	{attribute 'TcIecLibraryType'}
	{attribute 'external_name' := 'F_VN_CreateStaModel_GUID_E1160B26_F7CF_4D94_F7D4_A5AFD71C214D'}
	(* Create a Simplified TopoART neural network of the specified type. The initial reference count is set to one if a new model is created and kept, otherwise. Models of this type support on-line training (sample by sample), retraining, as well as scalar and vectorial predictions. It requires all input except class labels (i.e., samples and training outputs/predictions) to lie in the interval [0.0, 1.0]. The predictions of regressors need to be rescaled from the interval [0.0, 1.0] to their respective value range before usage. Depending on the parameter settings and the number of available training samples, repeated training with the same data may improve the results. Like other neural networks based on the Adaptive Resonance Theory (ART), Simplified TopoART neural networks are not prone to catastrophic inference and patricularly well-suited to incremental learning tasks. *)
	FUNCTION F_VN_CreateStaModel : HRESULT
	VAR_INPUT
		ipMlModel	:	REFERENCE TO ITcVnMlModel;	(* Returns the created model (Non-zero interface pointers are reused.) *)
		eStaType	:	ETcVnSta;	(* Simpified TopoART model type *)
		fRho	:	LREAL;	(* Vigilance parameter (controls the number of neurons that are inserted and the maximum size of the formed categories; valid range: [0.0, 1.0]; suggested range: [0.8, 1.0)) *)
		hrPrev	:	HRESULT;	(* HRESULT indicating the result of previous operations (If SUCCEEDED(hrPrev) equals false, no operation is executed.) *)
	END_VAR

END_FUNCTION

// Functions/Machine Learning/F_VN_CreateStaModelExp

	{attribute 'TcIecLibraryType'}
	{attribute 'external_name' := 'F_VN_CreateStaModelExp_GUID_8FBAA2F4_0437_4354_E26E_F8E69F80A9C2'}
	(* Create a Simplified TopoART neural network of the specified type. The initial reference count is set to one if a new model is created and kept, otherwise. Models of this type support on-line training (sample by sample), retraining, as well as scalar and vectorial predictions. It requires all input except class labels (i.e., samples and training outputs/predictions) to lie in the interval [0.0, 1.0]. The predictions of regressors need to be rescaled from the interval [0.0, 1.0] to their respective value range before usage. Depending on the parameter settings and the number of available training samples, repeated training with the same data may improve the results. Like other neural networks based on the Adaptive Resonance Theory (ART), Simplified TopoART neural networks are not prone to catastrophic inference and patricularly well-suited to incremental learning tasks. (expert function) *)
	FUNCTION F_VN_CreateStaModelExp : HRESULT
	VAR_INPUT
		ipMlModel	:	REFERENCE TO ITcVnMlModel;	(* Returns the created model (Non-zero interface pointers are reused.) *)
		eStaType	:	ETcVnSta;	(* Simpified TopoART model type *)
		fRho	:	LREAL;	(* Vigilance parameter (controls the number of neurons that are inserted and the maximum size of the formed categories; valid range: [0.0, 1.0]; suggested range: [0.8, 1.0)) *)
		nNu	:	UDINT;	(* Number of neurons used for classification and prediction (must be larger than or equal to 1; suggested range: [1, 10); default: 3) *)
		bDoublePrecision	:	BOOL;	(* If true, the model is generated with double precision (LREAL) instead of single precision (REAL). (default: FALSE) *)
		hrPrev	:	HRESULT;	(* HRESULT indicating the result of previous operations (If SUCCEEDED(hrPrev) equals false, no operation is executed.) *)
	END_VAR

END_FUNCTION

// Functions/Machine Learning/F_VN_CreateStaModelExp2

	{attribute 'TcIecLibraryType'}
	{attribute 'external_name' := 'F_VN_CreateStaModelExp2_GUID_332943B0_2083_4579_FA51_A2E1DF860F25'}
	(* Create a Simplified TopoART neural network of the specified type. The initial reference count is set to one if a new model is created and kept, otherwise. Models of this type support on-line training (sample by sample), retraining, as well as scalar and vectorial predictions. It requires all input except class labels (i.e., samples and training outputs/predictions) to lie in the interval [0.0, 1.0]. The predictions of regressors need to be rescaled from the interval [0.0, 1.0] to their respective value range before usage. Depending on the parameter settings and the number of available training samples, repeated training with the same data may improve the results. Like other neural networks based on the Adaptive Resonance Theory (ART), Simplified TopoART neural networks are not prone to catastrophic inference and patricularly well-suited to incremental learning tasks. (additional expert function providing parameters for fine-tuning and noise reduction) *)
	FUNCTION F_VN_CreateStaModelExp2 : HRESULT
	VAR_INPUT
		ipMlModel	:	REFERENCE TO ITcVnMlModel;	(* Returns the created model (Non-zero interface pointers are reused.) *)
		eStaType	:	ETcVnSta;	(* Simpified TopoART model type *)
		fRho	:	LREAL;	(* Vigilance parameter (controls the number of neurons that are inserted and the maximum size of the formed categories; valid range: [0.0, 1.0]; suggested range: [0.8, 1.0)) *)
		nNu	:	UDINT;	(* Number of neurons used for classification and prediction (must be larger than or equal to 1; suggested range: [1, 10); default: 3) *)
		bDoublePrecision	:	BOOL;	(* If true, the model is generated with double precision (LREAL) instead of single precision (REAL). (default: FALSE) *)
		fBetaSbm	:	LREAL;	(* Learning rate of the second best-matching neuron (learning the second best-matching neuron keeps related categories closer together and might improve the results but may require a higher number of neurons and training runs; a value of 0.0 disables learning of the second best-matching neuron; valid range: [0.0, 1.0]; suggested range: [0.0, 0.5]); default: 0.0 *)
		nPhi	:	UDINT;	(* Number of samples a neuron must have learnt to become permanent (required for noise reduction; works in conjunction with nTau; must be larger than or equal to 1; higher values intensify noise reduction; a value of 1 disables removal of neuron candidates; default: 1) *)
		nTau	:	UDINT;	(* Number of learning steps after which node removal is performed (required for noise reduction; works in conjunction with nPhi; must be large enough to allow neuron candidates representing non-noise samples to become the best-matching neuron at least nPhi times before node removal; default: 100) *)
		hrPrev	:	HRESULT;	(* HRESULT indicating the result of previous operations (If SUCCEEDED(hrPrev) equals false, no operation is executed.) *)
	END_VAR

END_FUNCTION

// Functions/Machine Learning/F_VN_CreateSvmModel

	{attribute 'TcIecLibraryType'}
	{attribute 'external_name' := 'F_VN_CreateSvmModel_GUID_897BE96D_4F53_4CE0_D9B9_89EE3A81129D'}
	(* Create an SVM model of the specified type. The initial reference count is set to one if a new model is created and kept, otherwise. Models of this type neither support on-line training (sample by sample) nor retraining. Predictions can only be scalar. *)
	FUNCTION F_VN_CreateSvmModel : HRESULT
	VAR_INPUT
		ipMlModel	:	REFERENCE TO ITcVnMlModel;	(* Returns the created model (Non-zero interface pointers are reused.) *)
		eSvmType	:	ETcVnSvm;	(* SVM model type *)
		fC	:	LREAL;	(* Parameter C (required for TCVN_SVM_C_CLASSIFIER, TCVN_SVM_EPS_REGRESSOR, and TCVN_SVM_NU_REGRESSOR; ignored otherwise) *)
		fNu	:	LREAL;	(* Parameter nu (required for TCVN_SVM_NU_CLASSIFIER, TCVN_SVM_NOVELTY_DETECTOR, and TCVN_SVM_NU_REGRESSOR; ignored otherwise) *)
		fP	:	LREAL;	(* Parameter p (required for TCVN_SVM_EPS_REGRESSOR; ignored otherwise) *)
		eKernelType	:	ETcVnSvmKernelType;	(* Kernel type *)
		fGamma	:	LREAL;	(* Parameter gamma (used by polynomial, RBF, sigmoid, and chi-squared kernels; ignored otherwise) *)
		fCoef0	:	LREAL;	(* parameter coef0 (used by polynomial and sigmoid kernels; ignored otherwise) *)
		fDegree	:	LREAL;	(* Degree (used by polynomial kernels; ignored otherwise) *)
		hrPrev	:	HRESULT;	(* HRESULT indicating the result of previous operations (If SUCCEEDED(hrPrev) equals false, no operation is executed.) *)
	END_VAR

END_FUNCTION

// Functions/Machine Learning/F_VN_CreateSvmModelExp

	{attribute 'TcIecLibraryType'}
	{attribute 'external_name' := 'F_VN_CreateSvmModelExp_GUID_846E7362_1CAD_446F_E876_9CE57F3D46D8'}
	(* Create an SVM model of the specified type. The initial reference count is set to one if a new model is created and kept, otherwise. Models of this type neither support on-line training (sample by sample) nor retraining. Predictions can only be scalar. (expert function) *)
	FUNCTION F_VN_CreateSvmModelExp : HRESULT
	VAR_INPUT
		ipMlModel	:	REFERENCE TO ITcVnMlModel;	(* Returns the created model (Non-zero interface pointers are reused.) *)
		eSvmType	:	ETcVnSvm;	(* SVM model type *)
		fC	:	LREAL;	(* Parameter C (required for TCVN_SVM_C_CLASSIFIER, TCVN_SVM_EPS_REGRESSOR, and TCVN_SVM_NU_REGRESSOR; ignored otherwise) *)
		fNu	:	LREAL;	(* Parameter nu (required for TCVN_SVM_NU_CLASSIFIER, TCVN_SVM_NOVELTY_DETECTOR, and TCVN_SVM_NU_REGRESSOR; ignored otherwise) *)
		fP	:	LREAL;	(* Parameter p (required for TCVN_SVM_EPS_REGRESSOR; ignored otherwise) *)
		eKernelType	:	ETcVnSvmKernelType;	(* Kernel type *)
		fGamma	:	LREAL;	(* Parameter gamma (used by polynomial, RBF, sigmoid, and chi-squared kernels; ignored otherwise) *)
		fCoef0	:	LREAL;	(* Parameter coef0 (used by polynomial and sigmoid kernels; ignored otherwise) *)
		fDegree	:	LREAL;	(* Degree (used by polynomial kernels; ignored otherwise) *)
		nMaxIterations	:	UDINT;	(* Maximum number of iterations (disabled if it equals 0 and fEpsilon is different from 0.0; triggers the usage of the default value of 100000 if nMaxIterations and fEpsilon equal 0) *)
		fEpsilon	:	LREAL;	(* Maximum allowed difference of the error between two successive iterations (disabled if it equals 0.0 and nMaxIterations is different from 0; triggers the usage of the default value of 0.00001 if nMaxIterations and fEpsilon equal 0) *)
		hrPrev	:	HRESULT;	(* HRESULT indicating the result of previous operations (If SUCCEEDED(hrPrev) equals false, no operation is executed.) *)
	END_VAR

END_FUNCTION

// Functions/Machine Learning/F_VN_CreateSvmModelExp2

	{attribute 'TcIecLibraryType'}
	{attribute 'external_name' := 'F_VN_CreateSvmModelExp2_GUID_80A60ED2_EC58_4E94_FB00_9F02BF868F8D'}
	(* Create an SVM model of the specified type. The initial reference count is set to one if a new model is created and kept, otherwise. Models of this type neither support on-line training (sample by sample) nor retraining. Predictions can only be scalar. (additional expert function for C support vector classifiers) *)
	FUNCTION F_VN_CreateSvmModelExp2 : HRESULT
	VAR_INPUT
		ipMlModel	:	REFERENCE TO ITcVnMlModel;	(* Returns the created model (Non-zero interface pointers are reused.) *)
		eSvmType	:	ETcVnSvm;	(* SVM model type *)
		fC	:	LREAL;	(* Parameter C (required for TCVN_SVM_C_CLASSIFIER, TCVN_SVM_EPS_REGRESSOR, and TCVN_SVM_NU_REGRESSOR; ignored otherwise) *)
		fNu	:	LREAL;	(* Parameter nu (required for TCVN_SVM_NU_CLASSIFIER, TCVN_SVM_NOVELTY_DETECTOR, and TCVN_SVM_NU_REGRESSOR; ignored otherwise) *)
		fP	:	LREAL;	(* Parameter p (required for TCVN_SVM_EPS_REGRESSOR; ignored otherwise) *)
		eKernelType	:	ETcVnSvmKernelType;	(* Kernel type *)
		fGamma	:	LREAL;	(* Parameter gamma (used by polynomial, RBF, sigmoid, and chi-squared kernels; ignored otherwise) *)
		fCoef0	:	LREAL;	(* Parameter coef0 (used by polynomial and sigmoid kernels; ignored otherwise) *)
		fDegree	:	LREAL;	(* Degree (used by polynomial kernels; ignored otherwise) *)
		nMaxIterations	:	UDINT;	(* Maximum number of iterations (disabled if it equals 0 and fEpsilon is different from 0.0; triggers the usage of the default value of 100000 if nMaxIterations and fEpsilon equal 0) *)
		fEpsilon	:	LREAL;	(* Maximum allowed difference of the error between two successive iterations (disabled if it equals 0.0 and nMaxIterations is different from 0; triggers the usage of the default value of 0.00001 if nMaxIterations and fEpsilon equal 0) *)
		ipClassWeights	:	ITcVnContainer;	(* Class weights (ContainerType_Vector_REAL or ContainerType_Vector_LREAL; only valid if eSvmType equals TCVN_SVM_C_CLASSIFIER; optional, set to 0 if not required or not allowed; default: 0) *)
		hrPrev	:	HRESULT;	(* HRESULT indicating the result of previous operations (If SUCCEEDED(hrPrev) equals false, no operation is executed.) *)
	END_VAR

END_FUNCTION

// Functions/Machine Learning/F_VN_CreateSvmSgdClassifier

	{attribute 'TcIecLibraryType'}
	{attribute 'external_name' := 'F_VN_CreateSvmSgdClassifier_GUID_269DD8EF_015C_48A4_C0CA_F5AB46B04256'}
	(* Create a linear SVM classifier using stochastic gradient descent for training. The initial reference count is set to one if a new model is created and kept, otherwise. This SVM classifier is only applicable to binary classification problems. It learns a separating hyperplane between a class with label -1 and a class with label 1. These class labels are predefined. For training, any positive class labels are mapped to 1 and any negative class labels are mapped to -1. Models of this type neither support on-line training (sample by sample) nor retraining. *)
	FUNCTION F_VN_CreateSvmSgdClassifier : HRESULT
	VAR_INPUT
		ipMlModel	:	REFERENCE TO ITcVnMlModel;	(* Returns the created model (Non-zero interface pointers are reused.) *)
		hrPrev	:	HRESULT;	(* HRESULT indicating the result of previous operations (If SUCCEEDED(hrPrev) equals false, no operation is executed.) *)
	END_VAR

END_FUNCTION

// Functions/Machine Learning/F_VN_CreateSvmSgdClassifierExp

	{attribute 'TcIecLibraryType'}
	{attribute 'external_name' := 'F_VN_CreateSvmSgdClassifierExp_GUID_DA02D1B9_7AEC_4B7E_EFA9_4DE4F7562F76'}
	(* Create a linear SVM classifier using stochastic gradient descent for training. The initial reference count is set to one if a new model is created and kept, otherwise. This SVM classifier is only applicable to binary classification problems. It learns a separating hyperplane between a class with label -1 and a class with label 1. These class labels are predefined. For training, any positive class labels are mapped to 1 and any negative class labels are mapped to -1. Models of this type neither support on-line training (sample by sample) nor retraining. (expert function) *)
	FUNCTION F_VN_CreateSvmSgdClassifierExp : HRESULT
	VAR_INPUT
		ipMlModel	:	REFERENCE TO ITcVnMlModel;	(* Returns the created model (Non-zero interface pointers are reused.) *)
		eType	:	ETcVnSvmSgdClassifierType;	(* Learning algorithm type (default: TCVN_SSCT_ASGD) *)
		eMarginType	:	ETcVnSvmSgdClassifierMarginType;	(* Margin type (default: TCVN_SSCMT_SOFT_MARGIN) *)
		fMarginRegularization	:	REAL;	(* Margin regularization parameter (default: 0.00001) *)
		fInitialStepSize	:	REAL;	(* Initial step size (default: 0.05) *)
		fStepDecreasingPower	:	REAL;	(* Power parameter (default: 0.75) *)
		nMaxIterations	:	UDINT;	(* Maximum number of iterations (disabled if it equals 0 and fEpsilon is different from 0.0; triggers the usage of the default value of 100000 if nMaxIterations and fEpsilon equal 0) *)
		fEpsilon	:	LREAL;	(* Maximum allowed difference of the error between two successive iterations (disabled if it equals 0.0 and nMaxIterations is different from 0; triggers the usage of the default value of 0.00001 if nMaxIterations and fEpsilon equal 0) *)
		hrPrev	:	HRESULT;	(* HRESULT indicating the result of previous operations (If SUCCEEDED(hrPrev) equals false, no operation is executed.) *)
	END_VAR

END_FUNCTION

// Functions/Machine Learning/F_VN_FeatureTransform

	{attribute 'TcIecLibraryType'}
	{attribute 'external_name' := 'F_VN_FeatureTransform_GUID_2974563E_7A4B_46F8_CDD5_2C6660AA8677'}
	(* Apply a feature transform to one or more sample(s). *)
	FUNCTION F_VN_FeatureTransform : HRESULT
	VAR_INPUT
		ipFeatureTransform	:	ITcVnMlModel;	(* Feature transform instance to be used *)
		ipSamples	:	ITcUnknown;	(* Container holding one or more of input sample(s) (ContainerType_Vector_REAL, ContainerType_Vector_LREAL, ContainerType_Vector_Vector_REAL, or ContainerType_Vector_Vector_LREAL) *)
		pipTransformed	:	POINTER TO ITcUnknown;	(* Returns the transformed sample(s) using the same type like ipSamples *)
		hrPrev	:	HRESULT;	(* HRESULT indicating the result of previous operations (If SUCCEEDED(hrPrev) equals false, no operation is executed.) *)
	END_VAR

END_FUNCTION

// Functions/Machine Learning/F_VN_GetBatchClusters

	{attribute 'TcIecLibraryType'}
	{attribute 'external_name' := 'F_VN_GetBatchClusters_GUID_BDFDD55D_49E0_4ED4_F9D7_56F0B43B3AD1'}
	(* Get the IDs of the best-matching clusters of a batch of samples. *)
	FUNCTION F_VN_GetBatchClusters : HRESULT
	VAR_INPUT
		ipClusterer	:	ITcVnMlModel;	(* Clusterer to be used *)
		ipSamples	:	ITcUnknown;	(* Container holding a batch of input samples (ContainerType_Vector_Vector_REAL or ContainerType_Vector_Vector_LREAL) *)
		ipClusters	:	REFERENCE TO ITcVnContainer;	(* Returns the cluster IDs (ContainerType_Vector_DINT) *)
		hrPrev	:	HRESULT;	(* HRESULT indicating the result of previous operations (If SUCCEEDED(hrPrev) equals false, no operation is executed.) *)
	END_VAR

END_FUNCTION

// Functions/Machine Learning/F_VN_GetBatchClustersExp

	{attribute 'TcIecLibraryType'}
	{attribute 'external_name' := 'F_VN_GetBatchClustersExp_GUID_05544234_9673_4981_C2EB_ED06839AEAC5'}
	(* Get the IDs of the best-matching clusters of a batch of samples. *)
	FUNCTION F_VN_GetBatchClustersExp : HRESULT
	VAR_INPUT
		ipClusterer	:	ITcVnMlModel;	(* Clusterer to be used *)
		ipSamples	:	ITcUnknown;	(* Container holding a batch of input samples (ContainerType_Vector_Vector_REAL or ContainerType_Vector_Vector_LREAL) *)
		ipClusters	:	REFERENCE TO ITcVnContainer;	(* Returns the cluster IDs (ContainerType_Vector_DINT) *)
		ipNovelties	:	REFERENCE TO ITcVnContainer;	(* Returns the degree of novelty (0.0 if a sample is completely known; > 0.0 otherwise) of each sample (ContainerType_Vector_REAL; optional, set to 0 if not required) *)
		hrPrev	:	HRESULT;	(* HRESULT indicating the result of previous operations (If SUCCEEDED(hrPrev) equals false, no operation is executed.) *)
	END_VAR

END_FUNCTION

// Functions/Machine Learning/F_VN_GetBatchNovelties

	{attribute 'TcIecLibraryType'}
	{attribute 'external_name' := 'F_VN_GetBatchNovelties_GUID_93485253_723B_43D7_F5BA_82F42BF1627D'}
	(* Get the degree of novelty of multiple samples. *)
	FUNCTION F_VN_GetBatchNovelties : HRESULT
	VAR_INPUT
		ipNoveltyDetector	:	ITcVnMlModel;	(* Novelty detector to be used *)
		ipSamples	:	ITcUnknown;	(* Container holding a batch of input samples (ContainerType_Vector_Vector_REAL or ContainerType_Vector_Vector_LREAL) *)
		ipNovelties	:	REFERENCE TO ITcVnContainer;	(* Returns the degree of novelty (0.0 if a sample is completely known; > 0.0 otherwise) of each sample (ContainerType_Vector_REAL) *)
		hrPrev	:	HRESULT;	(* HRESULT indicating the result of previous operations (If SUCCEEDED(hrPrev) equals false, no operation is executed.) *)
	END_VAR

END_FUNCTION

// Functions/Machine Learning/F_VN_GetClusterCenter

	{attribute 'TcIecLibraryType'}
	{attribute 'external_name' := 'F_VN_GetClusterCenter_GUID_E0FF4273_E499_42E6_FD8B_B6C189318933'}
	(* Get the center of a cluster. *)
	FUNCTION F_VN_GetClusterCenter : HRESULT
	VAR_INPUT
		ipClusterer	:	ITcVnMlModel;	(* Clusterer to be used *)
		nCluster	:	DINT;	(* Cluster ID of the cluster the center of which is requested *)
		ipCenter	:	REFERENCE TO ITcVnContainer;	(* Returns the cluster center (ContainerType_Vector_REAL or ContainerType_Vector_LREAL depending on the floating point type internally used by the clusterer) *)
		hrPrev	:	HRESULT;	(* HRESULT indicating the result of previous operations (If SUCCEEDED(hrPrev) equals false, no operation is executed.) *)
	END_VAR

END_FUNCTION

// Functions/Machine Learning/F_VN_GetClusterNum

	{attribute 'TcIecLibraryType'}
	{attribute 'external_name' := 'F_VN_GetClusterNum_GUID_BBFC8079_9A14_4919_DF9B_189A17F3D8B0'}
	(* Get the number of clusters used by this clusterer. *)
	FUNCTION F_VN_GetClusterNum : HRESULT
	VAR_INPUT
		ipClusterer	:	ITcVnMlModel;	(* Clusterer to be used *)
	END_VAR
	VAR_IN_OUT
		nClusterNum	:	ULINT;	(* Returns the number of clusters *)
	END_VAR
	VAR_INPUT
		hrPrev	:	HRESULT;	(* HRESULT indicating the result of previous operations (If SUCCEEDED(hrPrev) equals false, no operation is executed.) *)
	END_VAR

END_FUNCTION

// Functions/Machine Learning/F_VN_GetFeatureScales

	{attribute 'TcIecLibraryType'}
	{attribute 'external_name' := 'F_VN_GetFeatureScales_GUID_11456483_F148_42D1_FF0B_C79EBE00E4BF'}
	(* Calculate the scaling parameters for each feature in the input samples based on the scaling type. *)
	FUNCTION F_VN_GetFeatureScales : HRESULT
	VAR_INPUT
		ipSamples	:	ITcVnContainer;	(* Container holding input sample(s) (ContainerType_Vector_REAL, ContainerType_Vector_LREAL, ContainerType_Vector_Vector_REAL or ContainerType_Vector_Vector_LREAL) *)
		ipScales	:	REFERENCE TO ITcVnContainer;	(* Returns a container with the scaling parameters for each feature (Vector_REAL or Vector_LREAL depending on the type of ipSamples). *)
		eFeatureScalingType	:	ETcVnFeatureScalingType;	(* Feature scaling type *)
		hrPrev	:	HRESULT;	(* HRESULT indicating the result of previous operations (If SUCCEEDED(hrPrev) equals false, no operation is executed.) *)
	END_VAR

END_FUNCTION

// Functions/Machine Learning/F_VN_GetSampleCluster

	{attribute 'TcIecLibraryType'}
	{attribute 'external_name' := 'F_VN_GetSampleCluster_GUID_DD81FA91_6080_4B4C_E0CB_06C1EA1FBF26'}
	(* Get the ID of the best-matching cluster of a single sample. *)
	FUNCTION F_VN_GetSampleCluster : HRESULT
	VAR_INPUT
		ipClusterer	:	ITcVnMlModel;	(* Clusterer to be used *)
		ipSample	:	ITcUnknown;	(* Container holding a single input sample (ContainerType_Vector_REAL or ContainerType_Vector_LREAL) *)
	END_VAR
	VAR_IN_OUT
		nCluster	:	DINT;	(* Returns the ID of the cluster the sample has been assigned to *)
	END_VAR
	VAR_INPUT
		hrPrev	:	HRESULT;	(* HRESULT indicating the result of previous operations (If SUCCEEDED(hrPrev) equals false, no operation is executed.) *)
	END_VAR

END_FUNCTION

// Functions/Machine Learning/F_VN_GetSampleClusterExp

	{attribute 'TcIecLibraryType'}
	{attribute 'external_name' := 'F_VN_GetSampleClusterExp_GUID_DB048C2F_2D45_4057_FF4A_13B0418E387B'}
	(* Get the ID of the best-matching cluster of a single sample. (expert function) *)
	FUNCTION F_VN_GetSampleClusterExp : HRESULT
	VAR_INPUT
		ipClusterer	:	ITcVnMlModel;	(* Clusterer to be used *)
		ipSample	:	ITcUnknown;	(* Container holding a single input sample (ContainerType_Vector_REAL or ContainerType_Vector_LREAL) *)
	END_VAR
	VAR_IN_OUT
		nCluster	:	DINT;	(* Returns the ID of the cluster the sample has been assigned to *)
	END_VAR
	VAR_INPUT
		fNovelty	:	REFERENCE TO REAL;	(* Returns the degree of novelty (0.0 if a sample is completely known; > 0.0 otherwise) of the presented sample (optional, set to 0 if not required) *)
		hrPrev	:	HRESULT;	(* HRESULT indicating the result of previous operations (If SUCCEEDED(hrPrev) equals false, no operation is executed.) *)
	END_VAR

END_FUNCTION

// Functions/Machine Learning/F_VN_GetSampleNovelty

	{attribute 'TcIecLibraryType'}
	{attribute 'external_name' := 'F_VN_GetSampleNovelty_GUID_3DC424A1_B05C_4823_FDDB_8F0CF1505A59'}
	(* Get the degree of novelty of a single sample. *)
	FUNCTION F_VN_GetSampleNovelty : HRESULT
	VAR_INPUT
		ipNoveltyDetector	:	ITcVnMlModel;	(* Novelty detector to be used *)
		ipSample	:	ITcUnknown;	(* Container holding a single input sample (ContainerType_Vector_REAL or ContainerType_Vector_LREAL) *)
	END_VAR
	VAR_IN_OUT
		fNovelty	:	REAL;	(* Returns the degree of novelty (0.0 if a sample is completely known; > 0.0 otherwise) of the presented sample *)
	END_VAR
	VAR_INPUT
		hrPrev	:	HRESULT;	(* HRESULT indicating the result of previous operations (If SUCCEEDED(hrPrev) equals false, no operation is executed.) *)
	END_VAR

END_FUNCTION

// Functions/Machine Learning/F_VN_InverseFeatureScaling

	{attribute 'TcIecLibraryType'}
	{attribute 'external_name' := 'F_VN_InverseFeatureScaling_GUID_FAE38955_0DF9_4C1B_F986_91CF8149BAD2'}
	(* Apply the inverse of feature scaling to one or more sample(s). *)
	FUNCTION F_VN_InverseFeatureScaling : HRESULT
	VAR_INPUT
		ipSamples	:	ITcVnContainer;	(* Container holding one or more input sample(s) (ContainerType_Vector_REAL, ContainerType_Vector_LREAL, ContainerType_Vector_Vector_REAL, or ContainerType_Vector_Vector_LREAL) *)
		ipScales	:	ITcVnContainer;	(* Container with the scaling parameters of each feature (type ContainerType_Vector_REAL or ContainerType_Vector_LREAL). *)
		ipInverseSamples	:	REFERENCE TO ITcVnContainer;	(* Returns the inversed sample(s) using the scaling type and parameters of ipScales. It has the same type of ipSamples. If the same container ipSamples is used, the source data will be replaced. *)
		hrPrev	:	HRESULT;	(* HRESULT indicating the result of previous operations (If SUCCEEDED(hrPrev) equals false, no operation is executed.) *)
	END_VAR

END_FUNCTION

// Functions/Machine Learning/F_VN_InverseFeatureScaling_REAL

	{attribute 'TcIecLibraryType'}
	{attribute 'external_name' := 'F_VN_InverseFeatureScaling_REAL_GUID_166D968F_147A_4210_E12A_96ABB8210FC5'}
	(* Apply the inverse of feature scaling to a single value. *)
	FUNCTION F_VN_InverseFeatureScaling_REAL : HRESULT
	VAR_INPUT
		fSample	:	REAL;	(* Sample value *)
		ipScales	:	ITcVnContainer;	(* Container with the scaling parameters of each feature (type ContainerType_Vector_REAL or ContainerType_Vector_LREAL). *)
	END_VAR
	VAR_IN_OUT
		fInverseSample	:	REAL;	(* Returns the inversed sample. *)
	END_VAR
	VAR_INPUT
		hrPrev	:	HRESULT;	(* HRESULT indicating the result of previous operations (If SUCCEEDED(hrPrev) equals false, no operation is executed.) *)
	END_VAR

END_FUNCTION

// Functions/Machine Learning/F_VN_InverseFeatureScalingExp

	{attribute 'TcIecLibraryType'}
	{attribute 'external_name' := 'F_VN_InverseFeatureScalingExp_GUID_647DF1EC_D563_4098_CB76_97CF9047029E'}
	(* Apply the inverse of feature scaling to one or more sample(s). [fA, fB] should be used if the scaling has been performed using TCVN_FST1_MINMAX with a predetermined output range.. (expert function) *)
	FUNCTION F_VN_InverseFeatureScalingExp : HRESULT
	VAR_INPUT
		ipSamples	:	ITcVnContainer;	(* Container holding one or more input sample(s) (ContainerType_Vector_REAL, ContainerType_Vector_LREAL, ContainerType_Vector_Vector_REAL, or ContainerType_Vector_Vector_LREAL) *)
		ipScales	:	ITcVnContainer;	(* Container with the scaling parameters of each feature (type ContainerType_Vector_REAL or ContainerType_Vector_LREAL). *)
		ipInverseSamples	:	REFERENCE TO ITcVnContainer;	(* Returns the inversed sample(s) using the scaling type and parameters of ipScales. It has the same type of ipSamples. If the same container ipSamples is used, the source data will be replaced. *)
		fA	:	LREAL;	(* represents the lower bound of the range for TCVN_FST1_MINMAX *)
		fB	:	LREAL;	(* represents the upper bound of the range for TCVN_FST1_MINMAX *)
		hrPrev	:	HRESULT;	(* HRESULT indicating the result of previous operations (If SUCCEEDED(hrPrev) equals false, no operation is executed.) *)
	END_VAR

END_FUNCTION

// Functions/Machine Learning/F_VN_InverseFeatureScalingExp_REAL

	{attribute 'TcIecLibraryType'}
	{attribute 'external_name' := 'F_VN_InverseFeatureScalingExp_REAL_GUID_CDDB6A41_2C3B_42C5_C560_BF34481C5C25'}
	(* Apply the inverse of feature scaling to a single value. [fA, fB] should be used if the scaling has been performed using TCVN_FST1_MINMAX with a predetermined output range. *)
	FUNCTION F_VN_InverseFeatureScalingExp_REAL : HRESULT
	VAR_INPUT
		fSample	:	REAL;	(* Sample value *)
		ipScales	:	ITcVnContainer;	(* Container with the scaling parameters of each feature (type ContainerType_Vector_REAL or ContainerType_Vector_LREAL). *)
	END_VAR
	VAR_IN_OUT
		fInverseSample	:	REAL;	(* Returns the inversed sample. *)
	END_VAR
	VAR_INPUT
		fA	:	LREAL;	(* represents the lower bound of the range for TCVN_FST1_MINMAX *)
		fB	:	LREAL;	(* represents the upper bound of the range for TCVN_FST1_MINMAX *)
		hrPrev	:	HRESULT;	(* HRESULT indicating the result of previous operations (If SUCCEEDED(hrPrev) equals false, no operation is executed.) *)
	END_VAR

END_FUNCTION

// Functions/Machine Learning/F_VN_InverseFeatureTransform

	{attribute 'TcIecLibraryType'}
	{attribute 'external_name' := 'F_VN_InverseFeatureTransform_GUID_329639C8_477F_4462_EC9B_877837D05181'}
	(* Apply an inverse feature transform to one or more sample(s). *)
	FUNCTION F_VN_InverseFeatureTransform : HRESULT
	VAR_INPUT
		ipFeatureTransform	:	ITcVnMlModel;	(* Feature transform instance to be used *)
		ipSamples	:	ITcUnknown;	(* Container holding one or more of input sample(s) (ContainerType_Vector_REAL, ContainerType_Vector_LREAL, ContainerType_Vector_Vector_REAL, or ContainerType_Vector_Vector_LREAL) *)
		pipTransformed	:	POINTER TO ITcUnknown;	(* Returns the transformed sample(s) using the same type like ipSamples *)
		hrPrev	:	HRESULT;	(* HRESULT indicating the result of previous operations (If SUCCEEDED(hrPrev) equals false, no operation is executed.) *)
	END_VAR

END_FUNCTION

// Functions/Machine Learning/F_VN_PredictBatch

	{attribute 'TcIecLibraryType'}
	{attribute 'external_name' := 'F_VN_PredictBatch_GUID_7906A2A4_9C1A_4EB4_C744_43C3CB5A8C79'}
	(* Compute predictions for a batch of samples. *)
	FUNCTION F_VN_PredictBatch : HRESULT
	VAR_INPUT
		ipMlModel	:	ITcVnMlModel;	(* Classifier or regressor to be used *)
		ipSamples	:	ITcUnknown;	(* Container holding a batch of input samples (ContainerType_Vector_Vector_REAL or ContainerType_Vector_Vector_LREAL) *)
		ipPredictions	:	REFERENCE TO ITcVnContainer;	(* Returns the predicted outputs (depending on ipSamples; class labels (for classification, ContainerType_Vector_DINT) or real-valued predictions (for regression with scalar output, ContainerType_Vector_REAL or ContainerType_Vector_LREAL; for regression with vectorial output, ContainerType_Vector_Vector_REAL or ContainerType_Vector_Vector_LREAL)) *)
		hrPrev	:	HRESULT;	(* HRESULT indicating the result of previous operations (If SUCCEEDED(hrPrev) equals false, no operation is executed.) *)
	END_VAR

END_FUNCTION

// Functions/Machine Learning/F_VN_PredictBatchExp

	{attribute 'TcIecLibraryType'}
	{attribute 'external_name' := 'F_VN_PredictBatchExp_GUID_C7E3B96F_60A8_4AAD_F208_9E382A2099F8'}
	(* Compute predictions for a batch of samples. (expert function) *)
	FUNCTION F_VN_PredictBatchExp : HRESULT
	VAR_INPUT
		ipMlModel	:	ITcVnMlModel;	(* Classifier or regressor to be used *)
		ipSamples	:	ITcUnknown;	(* Container holding a batch of input samples (ContainerType_Vector_Vector_REAL or ContainerType_Vector_Vector_LREAL) *)
		ipPredictions	:	REFERENCE TO ITcVnContainer;	(* Returns the predicted outputs (depending on ipSamples; class labels (for classification, ContainerType_Vector_DINT) or real-valued predictions (for regression with scalar output, ContainerType_Vector_REAL or ContainerType_Vector_LREAL; for regression with vectorial output, ContainerType_Vector_Vector_REAL or ContainerType_Vector_Vector_LREAL)) *)
		ipNovelties	:	REFERENCE TO ITcVnContainer;	(* Returns the degree of novelty (0.0 if a sample is completely known; > 0.0 otherwise) of each sample (ContainerType_Vector_REAL; optional, set to 0 if not required) *)
		hrPrev	:	HRESULT;	(* HRESULT indicating the result of previous operations (If SUCCEEDED(hrPrev) equals false, no operation is executed.) *)
	END_VAR

END_FUNCTION

// Functions/Machine Learning/F_VN_PredictSampleClass

	{attribute 'TcIecLibraryType'}
	{attribute 'external_name' := 'F_VN_PredictSampleClass_GUID_4A7121E2_C40C_4D6B_D87B_86DF80F92135'}
	(* Classify a single sample. *)
	FUNCTION F_VN_PredictSampleClass : HRESULT
	VAR_INPUT
		ipClassifier	:	ITcVnMlModel;	(* Classifier to be used *)
		ipSample	:	ITcUnknown;	(* Container holding a single input sample (ContainerType_Vector_REAL or ContainerType_Vector_LREAL) *)
	END_VAR
	VAR_IN_OUT
		nClass	:	DINT;	(* Returns the classification result *)
	END_VAR
	VAR_INPUT
		hrPrev	:	HRESULT;	(* HRESULT indicating the result of previous operations (If SUCCEEDED(hrPrev) equals false, no operation is executed.) *)
	END_VAR

END_FUNCTION

// Functions/Machine Learning/F_VN_PredictSampleClassExp

	{attribute 'TcIecLibraryType'}
	{attribute 'external_name' := 'F_VN_PredictSampleClassExp_GUID_7E949930_4452_469B_E4D3_CE540860A53A'}
	(* Classify a single sample. (expert function) *)
	FUNCTION F_VN_PredictSampleClassExp : HRESULT
	VAR_INPUT
		ipClassifier	:	ITcVnMlModel;	(* Classifier to be used *)
		ipSample	:	ITcUnknown;	(* Container holding a single input sample (ContainerType_Vector_REAL or ContainerType_Vector_LREAL) *)
	END_VAR
	VAR_IN_OUT
		nClass	:	DINT;	(* Returns the classification result *)
	END_VAR
	VAR_INPUT
		fNovelty	:	REFERENCE TO REAL;	(* Returns the degree of novelty (0.0 if a sample is completely known; > 0.0 otherwise) of the presented sample (optional, set to 0 if not required) *)
		hrPrev	:	HRESULT;	(* HRESULT indicating the result of previous operations (If SUCCEEDED(hrPrev) equals false, no operation is executed.) *)
	END_VAR

END_FUNCTION

// Functions/Machine Learning/F_VN_PredictSampleScalar

	{attribute 'TcIecLibraryType'}
	{attribute 'external_name' := 'F_VN_PredictSampleScalar_GUID_A40A5FE6_578F_494C_E511_207CF80FE52D'}
	(* Compute a scalar prediction for a single sample. *)
	FUNCTION F_VN_PredictSampleScalar : HRESULT
	VAR_INPUT
		ipRegressor	:	ITcVnMlModel;	(* Regressor to be used *)
		ipSample	:	ITcUnknown;	(* Container holding a single input sample (ContainerType_Vector_REAL or ContainerType_Vector_LREAL) *)
	END_VAR
	VAR_IN_OUT
		fPrediction	:	REAL;	(* Returns the predicted output *)
	END_VAR
	VAR_INPUT
		hrPrev	:	HRESULT;	(* HRESULT indicating the result of previous operations (If SUCCEEDED(hrPrev) equals false, no operation is executed.) *)
	END_VAR

END_FUNCTION

// Functions/Machine Learning/F_VN_PredictSampleScalarExp

	{attribute 'TcIecLibraryType'}
	{attribute 'external_name' := 'F_VN_PredictSampleScalarExp_GUID_367E34F1_4772_4005_C610_209F58792692'}
	(* Compute a scalar prediction for a single sample. (expert function) *)
	FUNCTION F_VN_PredictSampleScalarExp : HRESULT
	VAR_INPUT
		ipRegressor	:	ITcVnMlModel;	(* Regressor to be used *)
		ipSample	:	ITcUnknown;	(* Container holding a single input sample (ContainerType_Vector_REAL or ContainerType_Vector_LREAL) *)
	END_VAR
	VAR_IN_OUT
		fPrediction	:	REAL;	(* Returns the predicted output *)
	END_VAR
	VAR_INPUT
		fNovelty	:	REFERENCE TO REAL;	(* Returns the degree of novelty (0.0 if a sample is completely known; > 0.0 otherwise) of the presented sample (optional, set to 0 if not required) *)
		hrPrev	:	HRESULT;	(* HRESULT indicating the result of previous operations (If SUCCEEDED(hrPrev) equals false, no operation is executed.) *)
	END_VAR

END_FUNCTION

// Functions/Machine Learning/F_VN_PredictSampleVector

	{attribute 'TcIecLibraryType'}
	{attribute 'external_name' := 'F_VN_PredictSampleVector_GUID_172DA4F7_FC29_4D5D_F84B_CCD2E6CC2758'}
	(* Compute a vectorial prediction for a single sample. *)
	FUNCTION F_VN_PredictSampleVector : HRESULT
	VAR_INPUT
		ipRegressor	:	ITcVnMlModel;	(* Regressor to be used *)
		ipSample	:	ITcUnknown;	(* Container holding a single input sample (ContainerType_Vector_REAL or ContainerType_Vector_LREAL) *)
		ipPrediction	:	REFERENCE TO ITcVnContainer;	(* Returns the predicted output (ContainerType_Vector_REAL or ContainerType_Vector_LREAL, depending on ipSample) *)
		hrPrev	:	HRESULT;	(* HRESULT indicating the result of previous operations (If SUCCEEDED(hrPrev) equals false, no operation is executed.) *)
	END_VAR

END_FUNCTION

// Functions/Machine Learning/F_VN_PredictSampleVectorExp

	{attribute 'TcIecLibraryType'}
	{attribute 'external_name' := 'F_VN_PredictSampleVectorExp_GUID_07735102_4AA2_46A6_C4D9_B15C63AD99B2'}
	(* Compute a vectorial prediction for a single sample. (expert function) *)
	FUNCTION F_VN_PredictSampleVectorExp : HRESULT
	VAR_INPUT
		ipRegressor	:	ITcVnMlModel;	(* Regressor to be used *)
		ipSample	:	ITcUnknown;	(* Container holding a single input sample (ContainerType_Vector_REAL or ContainerType_Vector_LREAL) *)
		ipPrediction	:	REFERENCE TO ITcVnContainer;	(* Returns the predicted output (ContainerType_Vector_REAL or ContainerType_Vector_LREAL, depending on ipSample) *)
		fNovelty	:	REFERENCE TO REAL;	(* Returns the degree of novelty (0.0 if a sample is completely known; > 0.0 otherwise) of the presented sample (optional, set to 0 if not required) *)
		hrPrev	:	HRESULT;	(* HRESULT indicating the result of previous operations (If SUCCEEDED(hrPrev) equals false, no operation is executed.) *)
	END_VAR

END_FUNCTION

// Functions/Machine Learning/F_VN_FeatureScaling

	{attribute 'TcIecLibraryType'}
	{attribute 'external_name' := 'F_VN_FeatureScaling_GUID_9FB5D54E_2B28_4BDC_DFDE_B62044F088AC'}
	(* Apply a feature scaling to one or more sample(s). *)
	FUNCTION F_VN_FeatureScaling : HRESULT
	VAR_INPUT
		ipSamples	:	ITcVnContainer;	(* Container holding one or more input sample(s) (ContainerType_Vector_REAL, ContainerType_Vector_LREAL, ContainerType_Vector_Vector_REAL, or ContainerType_Vector_Vector_LREAL) *)
		ipScales	:	ITcVnContainer;	(* Container with the scaling parameters of each feature (type ContainerType_Vector_REAL or ContainerType_Vector_LREAL). *)
		ipScaledSamples	:	REFERENCE TO ITcVnContainer;	(* Returns the scaled sample(s) using the same type like ipSamples. If the same container ipSamples is uesd, the source data will be replaced. *)
		hrPrev	:	HRESULT;	(* HRESULT indicating the result of previous operations (If SUCCEEDED(hrPrev) equals false, no operation is executed.) *)
	END_VAR

END_FUNCTION

// Functions/Machine Learning/F_VN_FeatureScalingExp

	{attribute 'TcIecLibraryType'}
	{attribute 'external_name' := 'F_VN_FeatureScalingExp_GUID_66B24BFE_9031_4553_F21F_FA0BBFFFF2B0'}
	(* Apply a feature scaling to one or more sample(s) and get output range between [fA, fB] in the case of TCVN_FST1_MINMAX.  (expert function) *)
	FUNCTION F_VN_FeatureScalingExp : HRESULT
	VAR_INPUT
		ipSamples	:	ITcVnContainer;	(* Container holding one or more input sample(s) (ContainerType_Vector_REAL, ContainerType_Vector_LREAL, ContainerType_Vector_Vector_REAL, or ContainerType_Vector_Vector_LREAL) *)
		ipScales	:	ITcVnContainer;	(* Container with the scaling parameters of each feature (type ContainerType_Vector_REAL or ContainerType_Vector_LREAL). *)
		ipScaledSamples	:	REFERENCE TO ITcVnContainer;	(* Returns the scaled sample(s) using the same type like ipSamples. If the same container ipSamples is uesd, the source data will be replaced. *)
		fA	:	LREAL;	(* represents the lower bound of the range for TCVN_FST1_MINMAX *)
		fB	:	LREAL;	(* represents the upper bound of the range for TCVN_FST1_MINMAX *)
		hrPrev	:	HRESULT;	(* HRESULT indicating the result of previous operations (If SUCCEEDED(hrPrev) equals false, no operation is executed.) *)
	END_VAR

END_FUNCTION

// Functions/Machine Learning/F_VN_TrainBatch

	{attribute 'TcIecLibraryType'}
	{attribute 'external_name' := 'F_VN_TrainBatch_GUID_73F82A21_79CD_4474_CA00_DD7E810BA348'}
	(* Train a classifier, a clusterer, a novelty detector, or a regressor with a batch of samples. On-line trainable models are trained once with each sample. Depending on the application and the number of available training samples, repeated training of such models with the same data may improve the results. *)
	FUNCTION F_VN_TrainBatch : HRESULT
	VAR_INPUT
		ipMlModel	:	ITcVnMlModel;	(* Classifier, clusterer, novelty detector, or regressor to be used *)
		ipSamples	:	ITcUnknown;	(* Container holding a batch of input samples (ContainerType_Vector_Vector_REAL or ContainerType_Vector_Vector_LREAL) *)
		ipOutputs	:	ITcVnContainer;	(* Class labels (for classification, ContainerType_Vector_DINT) or target outputs (for regression with scalar output, ContainerType_Vector_REAL or ContainerType_Vector_LREAL; for regression with vectorial output, ContainerType_Vector_Vector_REAL or ContainerType_Vector_Vector_LREAL) to be learnt (must be 0 for clusterers and for novelty detectors) *)
		hrPrev	:	HRESULT;	(* HRESULT indicating the result of previous operations (If SUCCEEDED(hrPrev) equals false, no operation is executed.) *)
	END_VAR

END_FUNCTION

// Functions/Machine Learning/F_VN_TrainBatchClusters

	{attribute 'TcIecLibraryType'}
	{attribute 'external_name' := 'F_VN_TrainBatchClusters_GUID_272ADC4A_55CD_40B4_F968_65B14199D4F5'}
	(* Train a clusterer with a batch of samples and return the IDs of the clusters the samples have been assigned to, if requested. On-line trainable clusterers are trained once with each sample. Depending on the application and the number of available training samples, repeated training of such models with the same data may improve the results. *)
	FUNCTION F_VN_TrainBatchClusters : HRESULT
	VAR_INPUT
		ipClusterer	:	ITcVnMlModel;	(* Clusterer to be used *)
		ipSamples	:	ITcUnknown;	(* Container holding a batch of input samples (ContainerType_Vector_Vector_REAL or ContainerType_Vector_Vector_LREAL) *)
		ipClusters	:	REFERENCE TO ITcVnContainer;	(* Returns the IDs of the clusters the samples have been assigned to (ContainerType_Vector_DINT; optional, set to 0 if not required) *)
		hrPrev	:	HRESULT;	(* HRESULT indicating the result of previous operations (If SUCCEEDED(hrPrev) equals false, no operation is executed.) *)
	END_VAR

END_FUNCTION

// Functions/Machine Learning/F_VN_TrainSample

	{attribute 'TcIecLibraryType'}
	{attribute 'external_name' := 'F_VN_TrainSample_GUID_6F6670E1_3692_44BE_FB06_674C6EFB3F43'}
	(* Train a clusterer or a novelty detector with a single sample. *)
	FUNCTION F_VN_TrainSample : HRESULT
	VAR_INPUT
		ipMlModel	:	ITcVnMlModel;	(* Clusterer or novelty detector to be used *)
		ipSample	:	ITcUnknown;	(* Container holding a single input sample (ContainerType_Vector_REAL or ContainerType_Vector_LREAL) *)
		hrPrev	:	HRESULT;	(* HRESULT indicating the result of previous operations (If SUCCEEDED(hrPrev) equals false, no operation is executed.) *)
	END_VAR

END_FUNCTION

// Functions/Machine Learning/F_VN_TrainSampleClass

	{attribute 'TcIecLibraryType'}
	{attribute 'external_name' := 'F_VN_TrainSampleClass_GUID_05A64E90_55FA_45CF_FDB8_2105F78E81D1'}
	(* Train a classifier with a single sample. *)
	FUNCTION F_VN_TrainSampleClass : HRESULT
	VAR_INPUT
		ipClassifier	:	ITcVnMlModel;	(* Classifier to be used *)
		ipSample	:	ITcUnknown;	(* Container holding a single input sample (ContainerType_Vector_REAL or ContainerType_Vector_LREAL) *)
		nClass	:	DINT;	(* Class label to be learnt *)
		hrPrev	:	HRESULT;	(* HRESULT indicating the result of previous operations (If SUCCEEDED(hrPrev) equals false, no operation is executed.) *)
	END_VAR

END_FUNCTION

// Functions/Machine Learning/F_VN_TrainSampleCluster

	{attribute 'TcIecLibraryType'}
	{attribute 'external_name' := 'F_VN_TrainSampleCluster_GUID_343E64C2_DE56_4145_F502_F352497DB18B'}
	(* Train a clusterer with a single sample and return the ID of the cluster the sample has been assigned to, if requested. The clusterer must be online trainable. *)
	FUNCTION F_VN_TrainSampleCluster : HRESULT
	VAR_INPUT
		ipClusterer	:	ITcVnMlModel;	(* Clusterer to be used *)
		ipSample	:	ITcUnknown;	(* Container holding a single input sample (ContainerType_Vector_REAL or ContainerType_Vector_LREAL) *)
		nCluster	:	REFERENCE TO DINT;	(* Returns the ID of the cluster the sample has been assigned to (If the pointer is 0, no cluster ID is requested.) *)
		hrPrev	:	HRESULT;	(* HRESULT indicating the result of previous operations (If SUCCEEDED(hrPrev) equals false, no operation is executed.) *)
	END_VAR

END_FUNCTION

// Functions/Machine Learning/F_VN_TrainSampleScalar

	{attribute 'TcIecLibraryType'}
	{attribute 'external_name' := 'F_VN_TrainSampleScalar_GUID_5CBD0285_80B0_4A96_F720_162C311C1FF3'}
	(* Train a regressor with a single sample and scalar output. *)
	FUNCTION F_VN_TrainSampleScalar : HRESULT
	VAR_INPUT
		ipRegressor	:	ITcVnMlModel;	(* Regressor to be used *)
		ipSample	:	ITcUnknown;	(* Container holding a single input sample (ContainerType_Vector_REAL or ContainerType_Vector_LREAL) *)
		fOutput	:	REAL;	(* Scalar output to be learnt *)
		hrPrev	:	HRESULT;	(* HRESULT indicating the result of previous operations (If SUCCEEDED(hrPrev) equals false, no operation is executed.) *)
	END_VAR

END_FUNCTION

// Functions/Machine Learning/F_VN_TrainSampleVector

	{attribute 'TcIecLibraryType'}
	{attribute 'external_name' := 'F_VN_TrainSampleVector_GUID_A5E64EDC_AD34_41AF_FAB6_19C619D724B8'}
	(* Train a regressor with a single sample and vectorial output. *)
	FUNCTION F_VN_TrainSampleVector : HRESULT
	VAR_INPUT
		ipRegressor	:	ITcVnMlModel;	(* Regressor to be used *)
		ipSample	:	ITcUnknown;	(* Container holding a single input sample (ContainerType_Vector_REAL or ContainerType_Vector_LREAL) *)
		ipOutput	:	ITcVnContainer;	(* Vectorial output to be learnt (ContainerType_Vector_REAL or ContainerType_Vector_LREAL) *)
		hrPrev	:	HRESULT;	(* HRESULT indicating the result of previous operations (If SUCCEEDED(hrPrev) equals false, no operation is executed.) *)
	END_VAR

END_FUNCTION

// Functions/Drawing/F_VN_DrawArrow

	{attribute 'TcIecLibraryType'}
	{attribute 'external_name' := 'F_VN_DrawArrow_GUID_219FAA59_40C2_4064_C408_565BDDFC528F'}
	(* Draw an arrowed line. *)
	FUNCTION F_VN_DrawArrow : HRESULT
	VAR_INPUT
		nX1	:	UDINT;	(* x coordinate of the start point *)
		nY1	:	UDINT;	(* y coordinate of the start point *)
		nX2	:	UDINT;	(* x coordinate of the end point *)
		nY2	:	UDINT;	(* y coordinate of the end point *)
		ipDestImage	:	ITcVnImage;	(* Destination image *)
	END_VAR
	VAR_IN_OUT
		aColor	:	TcVnVector4_LREAL;	(* Color *)
	END_VAR
	VAR_INPUT
		nThickness	:	DINT;	(* Line thickness *)
		bDoubleHead	:	BOOL;	(* To draw an arrow on each side of the line. *)
		hrPrev	:	HRESULT;	(* HRESULT indicating the result of previous operations (If SUCCEEDED(hrPrev) equals false, no operation is executed.) *)
	END_VAR

END_FUNCTION

// Functions/Drawing/F_VN_DrawArrow_TcVnVector4_DINT

	{attribute 'TcIecLibraryType'}
	{attribute 'external_name' := 'F_VN_DrawArrow_TcVnVector4_DINT_GUID_CD974053_3A84_4A78_FF52_9525307415ED'}
	(* Draw an arrowed line. *)
	FUNCTION F_VN_DrawArrow_TcVnVector4_DINT : HRESULT
	VAR_IN_OUT
		aLine	:	TcVnVector4_DINT;	(* The start and end point of a line segment [x1, y1, x2, y2] *)
	END_VAR
	VAR_INPUT
		ipDestImage	:	ITcVnImage;	(* Destination image *)
	END_VAR
	VAR_IN_OUT
		aColor	:	TcVnVector4_LREAL;	(* Color *)
	END_VAR
	VAR_INPUT
		nThickness	:	DINT;	(* Line thickness *)
		bDoubleHead	:	BOOL;	(* To draw an arrow on each side of the line. *)
		hrPrev	:	HRESULT;	(* HRESULT indicating the result of previous operations (If SUCCEEDED(hrPrev) equals false, no operation is executed.) *)
	END_VAR

END_FUNCTION

// Functions/Drawing/F_VN_DrawArrowExp

	{attribute 'TcIecLibraryType'}
	{attribute 'external_name' := 'F_VN_DrawArrowExp_GUID_9874EFD7_9D2C_4A6E_E29C_9A7DCBDB5A42'}
	(* Draws an arrowed line. (expert function) *)
	FUNCTION F_VN_DrawArrowExp : HRESULT
	VAR_INPUT
		nX1	:	UDINT;	(* x coordinate of the start point *)
		nY1	:	UDINT;	(* y coordinate of the start point *)
		nX2	:	UDINT;	(* x coordinate of the end point *)
		nY2	:	UDINT;	(* y coordinate of the end point *)
		ipDestImage	:	ITcVnImage;	(* Destination image *)
	END_VAR
	VAR_IN_OUT
		aColor	:	TcVnVector4_LREAL;	(* Color *)
	END_VAR
	VAR_INPUT
		nThickness	:	DINT;	(* Line thickness *)
		bDoubleHead	:	BOOL;	(* To draw an arrow on each side of the line. *)
		eLineType	:	ETcVnLineType;	(* Line type *)
		nShift	:	UDINT;	(* Fractional bits of the coordinates (bit shift) *)
		fTipLenght	:	LREAL;	(* Lenght of the arrow's tip as a fraction of the line's lenght *)
		hrPrev	:	HRESULT;	(* HRESULT indicating the result of previous operations (If SUCCEEDED(hrPrev) equals false, no operation is executed.) *)
	END_VAR

END_FUNCTION

// Functions/Drawing/F_VN_DrawArrowExp_TcVnVector4_DINT

	{attribute 'TcIecLibraryType'}
	{attribute 'external_name' := 'F_VN_DrawArrowExp_TcVnVector4_DINT_GUID_EB1F5363_59BE_442A_FA36_95178B47EBDC'}
	(* Draws an arrowed line. (expert function) *)
	FUNCTION F_VN_DrawArrowExp_TcVnVector4_DINT : HRESULT
	VAR_IN_OUT
		aLine	:	TcVnVector4_DINT;	(* The start and end point of a line segment [x1, y1, x2, y2] *)
	END_VAR
	VAR_INPUT
		ipDestImage	:	ITcVnImage;	(* Destination image *)
	END_VAR
	VAR_IN_OUT
		aColor	:	TcVnVector4_LREAL;	(* Color *)
	END_VAR
	VAR_INPUT
		nThickness	:	DINT;	(* Line thickness *)
		bDoubleHead	:	BOOL;	(* To draw an arrow on each side of the line. *)
		eLineType	:	ETcVnLineType;	(* Line type *)
		nShift	:	UDINT;	(* Fractional bits of the coordinates (bit shift) *)
		fTipLenght	:	LREAL;	(* Lenght of the arrow's tip as a fraction of the line's lenght *)
		hrPrev	:	HRESULT;	(* HRESULT indicating the result of previous operations (If SUCCEEDED(hrPrev) equals false, no operation is executed.) *)
	END_VAR

END_FUNCTION

// Functions/Drawing/F_VN_DrawCircle

	{attribute 'TcIecLibraryType'}
	{attribute 'external_name' := 'F_VN_DrawCircle_GUID_E54EF870_255A_4D91_CCEB_101D0778E80E'}
	(* Draws a circle. *)
	FUNCTION F_VN_DrawCircle : HRESULT
	VAR_INPUT
		nCenterX	:	UDINT;	(* x coordinate of the center *)
		nCenterY	:	UDINT;	(* y coordinate of the center *)
		nRadius	:	UDINT;	(* Radius *)
		ipDestImage	:	ITcVnImage;	(* Destination image *)
	END_VAR
	VAR_IN_OUT
		aColor	:	TcVnVector4_LREAL;	(* Color *)
	END_VAR
	VAR_INPUT
		nThickness	:	DINT;	(* Line thickness (if negative, the circle is filled) *)
		hrPrev	:	HRESULT;	(* HRESULT indicating the result of previous operations (If SUCCEEDED(hrPrev) equals false, no operation is executed.) *)
	END_VAR

END_FUNCTION

// Functions/Drawing/F_VN_DrawCircleExp

	{attribute 'TcIecLibraryType'}
	{attribute 'external_name' := 'F_VN_DrawCircleExp_GUID_EBF1C3F3_0B87_4735_E6BF_D00B09B46DB9'}
	(* Draws a circle. *)
	FUNCTION F_VN_DrawCircleExp : HRESULT
	VAR_INPUT
		nCenterX	:	UDINT;	(* x coordinate of the center *)
		nCenterY	:	UDINT;	(* y coordinate of the center *)
		nRadius	:	UDINT;	(* Radius *)
		ipDestImage	:	ITcVnImage;	(* Destination image *)
	END_VAR
	VAR_IN_OUT
		aColor	:	TcVnVector4_LREAL;	(* Color *)
	END_VAR
	VAR_INPUT
		nThickness	:	DINT;	(* Line thickness (if negative, the circle is filled) *)
		eLineType	:	ETcVnLineType;	(* Line type *)
		hrPrev	:	HRESULT;	(* HRESULT indicating the result of previous operations (If SUCCEEDED(hrPrev) equals false, no operation is executed.) *)
	END_VAR

END_FUNCTION

// Functions/Drawing/F_VN_DrawCircles

	{attribute 'TcIecLibraryType'}
	{attribute 'external_name' := 'F_VN_DrawCircles_GUID_13EAF35C_B06F_4815_C884_30D225E98417'}
	(* Draws circles. *)
	FUNCTION F_VN_DrawCircles : HRESULT
	VAR_INPUT
		ipCircles	:	ITcVnContainer;	(* Container with circles (ContainerType_Vector_TcVnVector3_REAL; Each container element contains the x coordinate of the circle center [0], the y coordinate of the circle center [1], and the radius [2].) *)
		nCircleIndex	:	DINT;	(* Index of a specific circle to be drawn (if negative, all circles within the container are drawn) *)
		ipDestImage	:	ITcVnImage;	(* Destination image *)
	END_VAR
	VAR_IN_OUT
		aColor	:	TcVnVector4_LREAL;	(* Color *)
	END_VAR
	VAR_INPUT
		nThickness	:	DINT;	(* Line thickness (if negative, the circle is filled) *)
		hrPrev	:	HRESULT;	(* HRESULT indicating the result of previous operations (If SUCCEEDED(hrPrev) equals false, no operation is executed.) *)
	END_VAR

END_FUNCTION

// Functions/Drawing/F_VN_DrawCirclesExp

	{attribute 'TcIecLibraryType'}
	{attribute 'external_name' := 'F_VN_DrawCirclesExp_GUID_4084C455_AE24_4B16_CD21_E442AAEA2A01'}
	(* Draws circles. (expert function) *)
	FUNCTION F_VN_DrawCirclesExp : HRESULT
	VAR_INPUT
		ipCircles	:	ITcVnContainer;	(* Container with circles (ContainerType_Vector_TcVnVector3_REAL; Each container element contains the x coordinate of the circle center [0], the y coordinate of the circle center [1], and the radius [2].) *)
		nCircleIndex	:	DINT;	(* Index of a specific circle to be drawn (if negative, all circles within the container are drawn) *)
		ipDestImage	:	ITcVnImage;	(* Destination image *)
	END_VAR
	VAR_IN_OUT
		aColor	:	TcVnVector4_LREAL;	(* Color *)
	END_VAR
	VAR_INPUT
		nThickness	:	DINT;	(* Line thickness (if negative, the circle is filled) *)
		eLineType	:	ETcVnLineType;	(* Line type *)
		hrPrev	:	HRESULT;	(* HRESULT indicating the result of previous operations (If SUCCEEDED(hrPrev) equals false, no operation is executed.) *)
	END_VAR

END_FUNCTION

// Functions/Drawing/F_VN_DrawCircularArc

	{attribute 'TcIecLibraryType'}
	{attribute 'external_name' := 'F_VN_DrawCircularArc_GUID_E25A37E1_93AB_4946_DDE0_DA467037DDBC'}
	(* Draws a circular arc. *)
	FUNCTION F_VN_DrawCircularArc : HRESULT
	VAR_IN_OUT
		stCircularArc	:	TcVnCircularArc;	(* Circular arc definition *)
	END_VAR
	VAR_INPUT
		ipDestImage	:	ITcVnImage;	(* Destination image *)
	END_VAR
	VAR_IN_OUT
		aColor	:	TcVnVector4_LREAL;	(* Color *)
	END_VAR
	VAR_INPUT
		nThickness	:	DINT;	(* Line thickness (if negative, the arc is filled) *)
		hrPrev	:	HRESULT;	(* HRESULT indicating the result of previous operations (If SUCCEEDED(hrPrev) equals false, no operation is executed.) *)
	END_VAR

END_FUNCTION

// Functions/Drawing/F_VN_DrawCircularArcExp

	{attribute 'TcIecLibraryType'}
	{attribute 'external_name' := 'F_VN_DrawCircularArcExp_GUID_D9B37CB2_BAE4_440C_C152_969A4B69D972'}
	(* Draws a circular arc. (expert function) *)
	FUNCTION F_VN_DrawCircularArcExp : HRESULT
	VAR_IN_OUT
		stCircularArc	:	TcVnCircularArc;	(* Circular arc definition *)
	END_VAR
	VAR_INPUT
		ipDestImage	:	ITcVnImage;	(* Destination image *)
	END_VAR
	VAR_IN_OUT
		aColor	:	TcVnVector4_LREAL;	(* Color *)
	END_VAR
	VAR_INPUT
		nThickness	:	DINT;	(* Line thickness (if negative, the arc is filled) *)
		eLineType	:	ETcVnLineType;	(* Line type *)
		hrPrev	:	HRESULT;	(* HRESULT indicating the result of previous operations (If SUCCEEDED(hrPrev) equals false, no operation is executed.) *)
	END_VAR

END_FUNCTION

// Functions/Drawing/F_VN_DrawComponents

	{attribute 'TcIecLibraryType'}
	{attribute 'external_name' := 'F_VN_DrawComponents_GUID_E9922499_BF1D_45AC_D80D_6B3535350DD3'}
	(* Draw the results of connected component function. *)
	FUNCTION F_VN_DrawComponents : HRESULT
	VAR_INPUT
		ipLabelImage	:	ITcVnImage;	(* Image contains labels for each pixel (1 channel DINT or UINT). *)
		nLabelID	:	DINT;	(* Value of a specific label to be drawn (if negative, all components within the image are drawn) *)
		ipDestImage	:	REFERENCE TO ITcVnImage;	(* Destination image (An appropriate image will be created if required. The output image is 1 or 3 channels USINT). *)
		bShowLabelID	:	BOOL;	(* Show label ID in the center of the component on the destination image *)
		hrPrev	:	HRESULT;	(* HRESULT indicating the result of previous operations (If SUCCEEDED(hrPrev) equals false, no operation is executed.) *)
	END_VAR

END_FUNCTION

// Functions/Drawing/F_VN_DrawComponentsExp

	{attribute 'TcIecLibraryType'}
	{attribute 'external_name' := 'F_VN_DrawComponentsExp_GUID_67F7A137_6C61_4D22_D78F_645CEAAA63A6'}
	(* Draw the results of connected component function. (expert function) *)
	FUNCTION F_VN_DrawComponentsExp : HRESULT
	VAR_INPUT
		ipLabelImage	:	ITcVnImage;	(* Image contains labels for each pixel (1 channel DINT or UINT). *)
		nLabelID	:	DINT;	(* Value of a specific label to be drawn (if negative, all components within the image are drawn) *)
		ipDestImage	:	REFERENCE TO ITcVnImage;	(* Destination image (An appropriate image will be created if required. The output image is 1 or 3 channels USINT). *)
		bShowLabelID	:	BOOL;	(* Show lable ID in the center of the component on the destination image *)
	END_VAR
	VAR_IN_OUT
		aColor	:	TcVnVector4_LREAL;	(* Color to draw the components (for {-1, -1, -1, -1}, a random color is chosen for each component) *)
	END_VAR
	VAR_INPUT
		nThickness	:	DINT;	(* Text line thickness *)
		fFontScale	:	LREAL;	(* Scaling factor for the text *)
		hrPrev	:	HRESULT;	(* HRESULT indicating the result of previous operations (If SUCCEEDED(hrPrev) equals false, no operation is executed.) *)
	END_VAR

END_FUNCTION

// Functions/Drawing/F_VN_DrawContours

	{attribute 'TcIecLibraryType'}
	{attribute 'external_name' := 'F_VN_DrawContours_GUID_BD96A0E1_088D_495C_DC88_0A1555E00AA4'}
	(* Draws a single point set or multiple point sets that are interpreted as contours. *)
	FUNCTION F_VN_DrawContours : HRESULT
	VAR_INPUT
		ipContours	:	ITcVnContainer;	(* Single contour (ContainerType_Vector_TcVnPoint2_DINT) or multiple contours (ContainerType_Vector_Vector_TcVnPoint2_DINT) *)
		nContourIndex	:	DINT;	(* Index of a specific contour to be drawn (if negative, all contours within the container are drawn) *)
		ipDestImage	:	ITcVnImage;	(* Destination image *)
	END_VAR
	VAR_IN_OUT
		aColor	:	TcVnVector4_LREAL;	(* Color *)
	END_VAR
	VAR_INPUT
		nThickness	:	DINT;	(* Line thickness (if negative, the contours are filled) *)
		hrPrev	:	HRESULT;	(* HRESULT indicating the result of previous operations (If SUCCEEDED(hrPrev) equals false, no operation is executed.) *)
	END_VAR

END_FUNCTION

// Functions/Drawing/F_VN_DrawContoursExp

	{attribute 'TcIecLibraryType'}
	{attribute 'external_name' := 'F_VN_DrawContoursExp_GUID_CEFBF024_BBCC_4DBE_C01D_8D086DC8267C'}
	(* Draws a single point set or multiple point sets that are interpreted as contours. (expert function) *)
	FUNCTION F_VN_DrawContoursExp : HRESULT
	VAR_INPUT
		ipContours	:	ITcVnContainer;	(* Single contour (ContainerType_Vector_TcVnPoint2_DINT) or multiple contours (ContainerType_Vector_Vector_TcVnPoint2_DINT) *)
		nContourIndex	:	DINT;	(* Index of a specific contour to be drawn (if negative, all contours within the container are drawn) *)
		ipDestImage	:	ITcVnImage;	(* Destination image *)
	END_VAR
	VAR_IN_OUT
		aColor	:	TcVnVector4_LREAL;	(* Color *)
	END_VAR
	VAR_INPUT
		nThickness	:	DINT;	(* Line thickness (if negative, the contours are filled) *)
		eLineType	:	ETcVnLineType;	(* Line type *)
		ipHierarchy	:	ITcVnContainer;	(* Contour hierarchy (ContainerType_Vector_TcVnVector4_DINT) *)
		nMaxLevel	:	DINT;	(* Maximum level of contours to be drawn *)
	END_VAR
	VAR_IN_OUT
		aOffset	:	TcVnPoint;	(* Offset by which every contour point is shifted *)
	END_VAR
	VAR_INPUT
		hrPrev	:	HRESULT;	(* HRESULT indicating the result of previous operations (If SUCCEEDED(hrPrev) equals false, no operation is executed.) *)
	END_VAR

END_FUNCTION

// Functions/Drawing/F_VN_DrawEllipse

	{attribute 'TcIecLibraryType'}
	{attribute 'external_name' := 'F_VN_DrawEllipse_GUID_348B0EA6_8D61_4699_CBAC_E9971A365AF6'}
	(* Draws an ellipse. *)
	FUNCTION F_VN_DrawEllipse : HRESULT
	VAR_IN_OUT
		stEllipse	:	TcVnRotatedRectangle;	(* Ellipse to be drawn (rotation angle in degrees) *)
	END_VAR
	VAR_INPUT
		ipDestImage	:	ITcVnImage;	(* Destination image *)
	END_VAR
	VAR_IN_OUT
		aColor	:	TcVnVector4_LREAL;	(* Color *)
	END_VAR
	VAR_INPUT
		nThickness	:	DINT;	(* Line thickness (if negative, the ellipse is filled) *)
		hrPrev	:	HRESULT;	(* HRESULT indicating the result of previous operations (If SUCCEEDED(hrPrev) equals false, no operation is executed.) *)
	END_VAR

END_FUNCTION

// Functions/Drawing/F_VN_DrawEllipseExp

	{attribute 'TcIecLibraryType'}
	{attribute 'external_name' := 'F_VN_DrawEllipseExp_GUID_C5879EEA_4F57_40F1_ED9B_B7DB43373126'}
	(* Draws an ellipse. (expert function) *)
	FUNCTION F_VN_DrawEllipseExp : HRESULT
	VAR_IN_OUT
		stEllipse	:	TcVnRotatedRectangle;	(* Ellipse to be drawn (rotation angle in degrees) *)
	END_VAR
	VAR_INPUT
		ipDestImage	:	ITcVnImage;	(* Destination image *)
	END_VAR
	VAR_IN_OUT
		aColor	:	TcVnVector4_LREAL;	(* Color *)
	END_VAR
	VAR_INPUT
		nThickness	:	DINT;	(* Line thickness (if negative, the ellipse is filled) *)
		eLineType	:	ETcVnLineType;	(* Line type *)
		hrPrev	:	HRESULT;	(* HRESULT indicating the result of previous operations (If SUCCEEDED(hrPrev) equals false, no operation is executed.) *)
	END_VAR

END_FUNCTION

// Functions/Drawing/F_VN_DrawKeypoints

	{attribute 'TcIecLibraryType'}
	{attribute 'external_name' := 'F_VN_DrawKeypoints_GUID_7CD843D3_4144_4284_C31E_4AA71D51FA08'}
	(* Draws the keypoints for visualization purpose. *)
	FUNCTION F_VN_DrawKeypoints : HRESULT
	VAR_INPUT
		ipSrcImage	:	ITcVnImage;	(* Source image (elements of type USINT) *)
		ipKeyPoints	:	ITcVnContainer;	(* Container with the keypoints (ContainerType_Vector_TcVnKeyPoint) *)
		ipDestImage	:	REFERENCE TO ITcVnImage;	(* Destination image (An appropriate color image will be created if required.) *)
		hrPrev	:	HRESULT;	(* HRESULT indicating the result of previous operations (If SUCCEEDED(hrPrev) equals false, no operation is executed.) *)
	END_VAR

END_FUNCTION

// Functions/Drawing/F_VN_DrawKeypointsExp

	{attribute 'TcIecLibraryType'}
	{attribute 'external_name' := 'F_VN_DrawKeypointsExp_GUID_D2F3CEBD_F7EE_4247_FEEE_921FEBF1519F'}
	(* Draws the keypoints for visualization purpose. (expert function) *)
	FUNCTION F_VN_DrawKeypointsExp : HRESULT
	VAR_INPUT
		ipSrcImage	:	ITcVnImage;	(* Source image (elements of type USINT) *)
		ipKeyPoints	:	ITcVnContainer;	(* Container with the keypoints (ContainerType_Vector_TcVnKeyPoint) *)
		ipDestImage	:	REFERENCE TO ITcVnImage;	(* Destination image (An appropriate color image will be created if required.) *)
	END_VAR
	VAR_IN_OUT
		aColor	:	TcVnVector4_LREAL;	(* Color to draw the keypoints (for {-1, -1, -1, -1}, a random color is chosen for each point) *)
	END_VAR
	VAR_INPUT
		eFlags	:	ETcVnDrawMatchesFlags;	(* A combination of flags to support overdrawing an existing destination image and/or drawing additional (Rich-)Keypoint information (size and orientation) *)
		hrPrev	:	HRESULT;	(* HRESULT indicating the result of previous operations (If SUCCEEDED(hrPrev) equals false, no operation is executed.) *)
	END_VAR

END_FUNCTION

// Functions/Drawing/F_VN_DrawLine

	{attribute 'TcIecLibraryType'}
	{attribute 'external_name' := 'F_VN_DrawLine_GUID_0270260A_8A1F_484E_F87D_D7BEE61DA000'}
	(* Draws a line. *)
	FUNCTION F_VN_DrawLine : HRESULT
	VAR_INPUT
		nX1	:	UDINT;	(* x coordinate of the start point *)
		nY1	:	UDINT;	(* y coordinate of the start point *)
		nX2	:	UDINT;	(* x coordinate of the end point *)
		nY2	:	UDINT;	(* y coordinate of the end point *)
		ipDestImage	:	ITcVnImage;	(* Destination image *)
	END_VAR
	VAR_IN_OUT
		aColor	:	TcVnVector4_LREAL;	(* Color *)
	END_VAR
	VAR_INPUT
		nThickness	:	DINT;	(* Line thickness *)
		hrPrev	:	HRESULT;	(* HRESULT indicating the result of previous operations (If SUCCEEDED(hrPrev) equals false, no operation is executed.) *)
	END_VAR

END_FUNCTION

// Functions/Drawing/F_VN_DrawLineExp

	{attribute 'TcIecLibraryType'}
	{attribute 'external_name' := 'F_VN_DrawLineExp_GUID_5A2061E8_A376_4B6D_D5EE_C02F1D812A9B'}
	(* Draws a line. (expert function) *)
	FUNCTION F_VN_DrawLineExp : HRESULT
	VAR_INPUT
		nX1	:	UDINT;	(* x coordinate of the start point *)
		nY1	:	UDINT;	(* y coordinate of the start point *)
		nX2	:	UDINT;	(* x coordinate of the end point *)
		nY2	:	UDINT;	(* y coordinate of the end point *)
		ipDestImage	:	ITcVnImage;	(* Destination image *)
	END_VAR
	VAR_IN_OUT
		aColor	:	TcVnVector4_LREAL;	(* Color *)
	END_VAR
	VAR_INPUT
		nThickness	:	DINT;	(* Line thickness *)
		eLineType	:	ETcVnLineType;	(* Line type *)
		nShift	:	UDINT;	(* Fractional bits of the coordinates (bit shift) *)
		hrPrev	:	HRESULT;	(* HRESULT indicating the result of previous operations (If SUCCEEDED(hrPrev) equals false, no operation is executed.) *)
	END_VAR

END_FUNCTION

// Functions/Drawing/F_VN_DrawLine_TcVnVector4_DINT

	{attribute 'TcIecLibraryType'}
	{attribute 'external_name' := 'F_VN_DrawLine_TcVnVector4_DINT_GUID_8C2ADBD1_2AAC_4B5A_F959_A826E5034260'}
	(* Draws a line. *)
	FUNCTION F_VN_DrawLine_TcVnVector4_DINT : HRESULT
	VAR_IN_OUT
		aLine	:	TcVnVector4_DINT;	(* The start and end point of a line segment [x1, y1, x2, y2] *)
	END_VAR
	VAR_INPUT
		ipDestImage	:	ITcVnImage;	(* Destination image *)
	END_VAR
	VAR_IN_OUT
		aColor	:	TcVnVector4_LREAL;	(* Color *)
	END_VAR
	VAR_INPUT
		nThickness	:	DINT;	(* Line thickness *)
		hrPrev	:	HRESULT;	(* HRESULT indicating the result of previous operations (If SUCCEEDED(hrPrev) equals false, no operation is executed.) *)
	END_VAR

END_FUNCTION

// Functions/Drawing/F_VN_DrawLineExp_TcVnVector4_DINT

	{attribute 'TcIecLibraryType'}
	{attribute 'external_name' := 'F_VN_DrawLineExp_TcVnVector4_DINT_GUID_EC4486FD_CFF6_4316_F560_A40C39451566'}
	(* Draws a line. (expert function) *)
	FUNCTION F_VN_DrawLineExp_TcVnVector4_DINT : HRESULT
	VAR_IN_OUT
		aLine	:	TcVnVector4_DINT;	(* The start and end point of a line segment [x1, y1, x2, y2] *)
	END_VAR
	VAR_INPUT
		ipDestImage	:	ITcVnImage;	(* Destination image *)
	END_VAR
	VAR_IN_OUT
		aColor	:	TcVnVector4_LREAL;	(* Color *)
	END_VAR
	VAR_INPUT
		nThickness	:	DINT;	(* Line thickness *)
		eLineType	:	ETcVnLineType;	(* Line type *)
		nShift	:	UDINT;	(* Fractional bits of the coordinates (bit shift) *)
		hrPrev	:	HRESULT;	(* HRESULT indicating the result of previous operations (If SUCCEEDED(hrPrev) equals false, no operation is executed.) *)
	END_VAR

END_FUNCTION

// Functions/Drawing/F_VN_DrawLine_TcVnVector4_LREAL

	{attribute 'TcIecLibraryType'}
	{attribute 'external_name' := 'F_VN_DrawLine_TcVnVector4_LREAL_GUID_77F4932D_ADE4_429C_C251_5C6A03CC1E85'}
	(* Draws a line. *)
	FUNCTION F_VN_DrawLine_TcVnVector4_LREAL : HRESULT
	VAR_IN_OUT
		aLine	:	TcVnVector4_LREAL;	(* The first and second element describe the x and y component of the direction vector. The third and fourth element describe the x and y component of the position vector. *)
	END_VAR
	VAR_INPUT
		ipDestImage	:	ITcVnImage;	(* Destination image *)
	END_VAR
	VAR_IN_OUT
		aColor	:	TcVnVector4_LREAL;	(* Color *)
	END_VAR
	VAR_INPUT
		nThickness	:	DINT;	(* Line thickness *)
		hrPrev	:	HRESULT;	(* HRESULT indicating the result of previous operations (If SUCCEEDED(hrPrev) equals false, no operation is executed.) *)
	END_VAR

END_FUNCTION

// Functions/Drawing/F_VN_DrawLineExp_TcVnVector4_LREAL

	{attribute 'TcIecLibraryType'}
	{attribute 'external_name' := 'F_VN_DrawLineExp_TcVnVector4_LREAL_GUID_CE9D84EC_5E0B_43AA_C118_9888CBF84588'}
	(* Draws a line. (expert function) *)
	FUNCTION F_VN_DrawLineExp_TcVnVector4_LREAL : HRESULT
	VAR_IN_OUT
		aLine	:	TcVnVector4_LREAL;	(* The first and second element describe the x and y component of the direction vector. The third and fourth element describe the x and y component of the position vector. *)
	END_VAR
	VAR_INPUT
		ipDestImage	:	ITcVnImage;	(* Destination image *)
	END_VAR
	VAR_IN_OUT
		aColor	:	TcVnVector4_LREAL;	(* Color *)
	END_VAR
	VAR_INPUT
		nThickness	:	DINT;	(* Line thickness *)
		eLineType	:	ETcVnLineType;	(* Line type *)
		nShift	:	UDINT;	(* Fractional bits of the coordinates (bit shift) *)
		hrPrev	:	HRESULT;	(* HRESULT indicating the result of previous operations (If SUCCEEDED(hrPrev) equals false, no operation is executed.) *)
	END_VAR

END_FUNCTION

// Functions/Drawing/F_VN_DrawLines

	{attribute 'TcIecLibraryType'}
	{attribute 'external_name' := 'F_VN_DrawLines_GUID_F81750F9_73FB_4365_C728_B3FCE8EC26AD'}
	(* Draws lines. *)
	FUNCTION F_VN_DrawLines : HRESULT
	VAR_INPUT
		ipLines	:	ITcVnContainer;	(* Container with line descriptions (ContainerType_Vector_TcVnVector2_REAL: the distance from the origin [0] in pixels and the rotation angle [1] in radians. ContainerType_Vector_TcVnVector4_LREAL: the first and second element describe the x and y component of a vector collinear to the line. The third and fourth element describe the x and y component of a point on the line. ContainerType_Vector_TcVnVector4_DINT: start and end point [x1, y1, x2, y2]) *)
		nLineIndex	:	DINT;	(* Index of a specific line to be drawn (if negative, all lines within the container are drawn) *)
		ipDestImage	:	ITcVnImage;	(* Destination image *)
	END_VAR
	VAR_IN_OUT
		aColor	:	TcVnVector4_LREAL;	(* Color *)
	END_VAR
	VAR_INPUT
		nThickness	:	DINT;	(* Line thickness *)
		hrPrev	:	HRESULT;	(* HRESULT indicating the result of previous operations (If SUCCEEDED(hrPrev) equals false, no operation is executed.) *)
	END_VAR

END_FUNCTION

// Functions/Drawing/F_VN_DrawLinesExp

	{attribute 'TcIecLibraryType'}
	{attribute 'external_name' := 'F_VN_DrawLinesExp_GUID_C304F022_2C45_4232_D759_3C25A105AD9F'}
	(* Draws lines. (expert function) *)
	FUNCTION F_VN_DrawLinesExp : HRESULT
	VAR_INPUT
		ipLines	:	ITcVnContainer;	(* Container with line descriptions (ContainerType_Vector_TcVnVector2_REAL: the distance from the origin [0] in pixels and the rotation angle [1] in radians. ContainerType_Vector_TcVnVector4_LREAL: the first and second element describe the x and y component of a vector collinear to the line. The third and fourth element describe the x and y component of a point on the line. ContainerType_Vector_TcVnVector4_DINT: start and end point [x1, y1, x2, y2]) *)
		nLineIndex	:	DINT;	(* Index of a specific line to be drawn (if negative, all lines within the container are drawn) *)
		ipDestImage	:	ITcVnImage;	(* Destination image *)
	END_VAR
	VAR_IN_OUT
		aColor	:	TcVnVector4_LREAL;	(* Color *)
	END_VAR
	VAR_INPUT
		nThickness	:	DINT;	(* Line thickness *)
		eLineType	:	ETcVnLineType;	(* Line type *)
		nShift	:	UDINT;	(* Fractional bits of the coordinates (bit shift) *)
		hrPrev	:	HRESULT;	(* HRESULT indicating the result of previous operations (If SUCCEEDED(hrPrev) equals false, no operation is executed.) *)
	END_VAR

END_FUNCTION

// Functions/Drawing/F_VN_DrawMatches

	{attribute 'TcIecLibraryType'}
	{attribute 'external_name' := 'F_VN_DrawMatches_GUID_13CA7DBE_CD1F_42F8_EDCC_81AEBD1E8357'}
	(* Draws the keypoints and matches for visualization purpose. *)
	FUNCTION F_VN_DrawMatches : HRESULT
	VAR_INPUT
		ipSrcImage1	:	ITcVnImage;	(* Source image 1 (elements of type USINT) *)
		ipKeyPoints1	:	ITcVnContainer;	(* Container with the keypoints 1 (ContainerType_Vector_TcVnKeyPoint) *)
		ipSrcImage2	:	ITcVnImage;	(* Source image 2 (elements of type USINT, must have the same number of channels as ipSrcImage1) *)
		ipKeyPoints2	:	ITcVnContainer;	(* Container with the keypoints 2 (ContainerType_Vector_TcVnKeyPoint) *)
		ipMatches1To2	:	ITcVnContainer;	(* Container with the descriptor matches (ContainerType_Vector_TcVnDMatch) *)
		ipDestImage	:	REFERENCE TO ITcVnImage;	(* Destination image (An appropriate color image will be created if required.) *)
		hrPrev	:	HRESULT;	(* HRESULT indicating the result of previous operations (If SUCCEEDED(hrPrev) equals false, no operation is executed.) *)
	END_VAR

END_FUNCTION

// Functions/Drawing/F_VN_DrawMatchesExp

	{attribute 'TcIecLibraryType'}
	{attribute 'external_name' := 'F_VN_DrawMatchesExp_GUID_59731CD6_4B44_4228_F527_D4613D090FCC'}
	(* Draws the keypoints and matches for visualization purpose. (expert function) *)
	FUNCTION F_VN_DrawMatchesExp : HRESULT
	VAR_INPUT
		ipSrcImage1	:	ITcVnImage;	(* Source image 1 (elements of type USINT) *)
		ipKeyPoints1	:	ITcVnContainer;	(* Container with the keypoints 1 (ContainerType_Vector_TcVnKeyPoint) *)
		ipSrcImage2	:	ITcVnImage;	(* Source image 2 (elements of type USINT, must have the same number of channels as ipSrcImage1) *)
		ipKeyPoints2	:	ITcVnContainer;	(* Container with the keypoints 2 (ContainerType_Vector_TcVnKeyPoint) *)
		ipMatches1To2	:	ITcVnContainer;	(* Container with the descriptor matches (ContainerType_Vector_TcVnDMatch) *)
		ipDestImage	:	REFERENCE TO ITcVnImage;	(* Destination image (An appropriate color image will be created if required.) *)
	END_VAR
	VAR_IN_OUT
		aMatchColor	:	TcVnVector4_LREAL;	(* Color to draw the matches (for {-1, -1, -1, -1}, a random color is chosen for each point and line) *)
		aSingleColor	:	TcVnVector4_LREAL;	(* Color to draw the single keypoints (for {-1, -1, -1, -1}, a random color is chosen for each point) *)
	END_VAR
	VAR_INPUT
		ipMatchesMask	:	ITcVnContainer;	(* Mask to select the matches to be drawn (ContainerType_Vector_SINT; Set to 0 if all matches should be drawn.) *)
		eFlags	:	ETcVnDrawMatchesFlags;	(* A combination of flags to support overdrawing an existing destination image and/or drawing additional (Rich-)Keypoint information (size and orientation) and/or skipping single keypoints *)
		hrPrev	:	HRESULT;	(* HRESULT indicating the result of previous operations (If SUCCEEDED(hrPrev) equals false, no operation is executed.) *)
	END_VAR

END_FUNCTION

// Functions/Drawing/F_VN_DrawOrientation

	{attribute 'TcIecLibraryType'}
	{attribute 'external_name' := 'F_VN_DrawOrientation_GUID_13B1D813_3D8E_47D6_F6E8_82EBE561B9DA'}
	(* Draw the main axis of a set of points/contour based on a rotated rectangle. *)
	FUNCTION F_VN_DrawOrientation : HRESULT
	VAR_IN_OUT
		stOrientation	:	TcVnRotatedRectangle;	(* Rotated rectangle, containig center of mass, lenghts of axes, and rotation angle in clockwise direction *)
	END_VAR
	VAR_INPUT
		ipDestImage	:	ITcVnImage;	(* Destination image *)
	END_VAR
	VAR_IN_OUT
		aColorMainAxis	:	TcVnVector4_LREAL;	(* Color of the major axis *)
	END_VAR
	VAR_INPUT
		nThickness	:	DINT;	(* Line thickness *)
		hrPrev	:	HRESULT;	(* HRESULT indicating the result of previous operations (If SUCCEEDED(hrPrev) equals false, no operation is executed.) *)
	END_VAR

END_FUNCTION

// Functions/Drawing/F_VN_DrawOrientationExp

	{attribute 'TcIecLibraryType'}
	{attribute 'external_name' := 'F_VN_DrawOrientationExp_GUID_F681A0E7_3FF2_4D39_C2E5_6D8D9C9B0334'}
	(* Draw the main axis, the horizontal axis and the angle of a set of points/contour based on a rotated rectangle. (expert function) *)
	FUNCTION F_VN_DrawOrientationExp : HRESULT
	VAR_IN_OUT
		stOrientation	:	TcVnRotatedRectangle;	(* Rotated rectangle, containig center of mass, lenghts of axes, and rotation angle in clockwise direction *)
	END_VAR
	VAR_INPUT
		ipDestImage	:	ITcVnImage;	(* Destination image *)
	END_VAR
	VAR_IN_OUT
		aColorMainAxis	:	TcVnVector4_LREAL;	(* Color of the major axis *)
	END_VAR
	VAR_INPUT
		nThickness	:	DINT;	(* Line thickness *)
	END_VAR
	VAR_IN_OUT
		aColorHorizontalAxis	:	TcVnVector4_LREAL;	(* Color of the horizontal axis *)
	END_VAR
	VAR_INPUT
		fFontScale	:	LREAL;	(* Scaling factor for the text *)
		hrPrev	:	HRESULT;	(* HRESULT indicating the result of previous operations (If SUCCEEDED(hrPrev) equals false, no operation is executed.) *)
	END_VAR

END_FUNCTION

// Functions/Drawing/F_VN_DrawPoint

	{attribute 'TcIecLibraryType'}
	{attribute 'external_name' := 'F_VN_DrawPoint_GUID_74F46D70_BCCE_44BB_D718_B65028EEE394'}
	(* Draws a point. *)
	FUNCTION F_VN_DrawPoint : HRESULT
	VAR_INPUT
		nX	:	UDINT;	(* x coordinate of the point *)
		nY	:	UDINT;	(* y coordinate of the point *)
		ipDestImage	:	ITcVnImage;	(* Destination image *)
		eShape	:	ETcVnDrawShape;	(* Point shape *)
	END_VAR
	VAR_IN_OUT
		aColor	:	TcVnVector4_LREAL;	(* Color (for {-1, -1, -1, -1}, a random color is chosen) *)
	END_VAR
	VAR_INPUT
		hrPrev	:	HRESULT;	(* HRESULT indicating the result of previous operations (If SUCCEEDED(hrPrev) equals false, no operation is executed.) *)
	END_VAR

END_FUNCTION

// Functions/Drawing/F_VN_DrawPointExp

	{attribute 'TcIecLibraryType'}
	{attribute 'external_name' := 'F_VN_DrawPointExp_GUID_935CF92C_D227_4D01_E807_8E54723B2E27'}
	(* Draw a point. (expert function) *)
	FUNCTION F_VN_DrawPointExp : HRESULT
	VAR_INPUT
		nX	:	UDINT;	(* x coordinate of the point *)
		nY	:	UDINT;	(* y coordinate of the point *)
		ipDestImage	:	ITcVnImage;	(* Destination image *)
		eShape	:	ETcVnDrawShape;	(* Point shape *)
	END_VAR
	VAR_IN_OUT
		aColor	:	TcVnVector4_LREAL;	(* Color (for {-1, -1, -1, -1}, a random color is chosen) *)
	END_VAR
	VAR_INPUT
		nSize	:	UDINT;	(* Size of the shape (half width) *)
		nThickness	:	DINT;	(* Line thickness (if negative, the shape is filled if it is closed) *)
		eLineType	:	ETcVnLineType;	(* Line type *)
		hrPrev	:	HRESULT;	(* HRESULT indicating the result of previous operations (If SUCCEEDED(hrPrev) equals false, no operation is executed.) *)
	END_VAR

END_FUNCTION

// Functions/Drawing/F_VN_DrawPoints

	{attribute 'TcIecLibraryType'}
	{attribute 'external_name' := 'F_VN_DrawPoints_GUID_79252F35_DEF8_4DE3_FEAD_58F3B9D6E295'}
	(* Draw a collection of points. *)
	FUNCTION F_VN_DrawPoints : HRESULT
	VAR_INPUT
		ipPoints	:	ITcVnContainer;	(* Container with TcVnPoint2_DINT or TcVnPoint2_REAL elements *)
		ipDestImage	:	ITcVnImage;	(* Destination image *)
		eShape	:	ETcVnDrawShape;	(* Point shape *)
	END_VAR
	VAR_IN_OUT
		aColor	:	TcVnVector4_LREAL;	(* Color (for {-1, -1, -1, -1}, a random color is chosen for each point) *)
	END_VAR
	VAR_INPUT
		hrPrev	:	HRESULT;	(* HRESULT indicating the result of previous operations (If SUCCEEDED(hrPrev) equals false, no operation is executed.) *)
	END_VAR

END_FUNCTION

// Functions/Drawing/F_VN_DrawPointsExp

	{attribute 'TcIecLibraryType'}
	{attribute 'external_name' := 'F_VN_DrawPointsExp_GUID_AB5F80E1_D173_4F9D_EE5F_B91F79CCBC5C'}
	(* Draw a collection of points. (expert function) *)
	FUNCTION F_VN_DrawPointsExp : HRESULT
	VAR_INPUT
		ipPoints	:	ITcVnContainer;	(* Container with TcVnPoint2_DINT or TcVnPoint2_REAL elements *)
		ipDestImage	:	ITcVnImage;	(* Destination image *)
		eShape	:	ETcVnDrawShape;	(* Point shape *)
	END_VAR
	VAR_IN_OUT
		aColor	:	TcVnVector4_LREAL;	(* Color (for {-1, -1, -1, -1}, a random color is chosen for each point) *)
	END_VAR
	VAR_INPUT
		nSize	:	UDINT;	(* Size of the shape (half width) *)
		nThickness	:	DINT;	(* Line thickness (if negative, the shape is filled if it is closed) *)
		eLineType	:	ETcVnLineType;	(* Line type *)
		hrPrev	:	HRESULT;	(* HRESULT indicating the result of previous operations (If SUCCEEDED(hrPrev) equals false, no operation is executed.) *)
	END_VAR

END_FUNCTION

// Functions/Drawing/F_VN_DrawPolygon

	{attribute 'TcIecLibraryType'}
	{attribute 'external_name' := 'F_VN_DrawPolygon_GUID_B52EC0EA_DC22_4E64_EBA7_6FFBA7400232'}
	(* Draw a pologon using collection of points. *)
	FUNCTION F_VN_DrawPolygon : HRESULT
	VAR_INPUT
		ipPoints	:	ITcVnContainer;	(* Container with TcVnPoint2_DINT, TcVnPoint2_REAL, or TcVnPoint2_LREAL elements *)
		ipDestImage	:	ITcVnImage;	(* Destination image *)
	END_VAR
	VAR_IN_OUT
		aColor	:	TcVnVector4_LREAL;	(* Color *)
	END_VAR
	VAR_INPUT
		nThickness	:	DINT;	(* Line thickness (if negative, the polygon is filled) *)
		hrPrev	:	HRESULT;	(* HRESULT indicating the result of previous operations (If SUCCEEDED(hrPrev) equals false, no operation is executed.) *)
	END_VAR

END_FUNCTION

// Functions/Drawing/F_VN_DrawPolygonExp

	{attribute 'TcIecLibraryType'}
	{attribute 'external_name' := 'F_VN_DrawPolygonExp_GUID_487782DD_5E9A_426D_E457_2C3350E60D47'}
	(* Draw a pologon using collection of points. (expert function) *)
	FUNCTION F_VN_DrawPolygonExp : HRESULT
	VAR_INPUT
		ipPoints	:	ITcVnContainer;	(* Container with TcVnPoint2_DINT, TcVnPoint2_REAL, or TcVnPoint2_LREAL elements *)
		ipDestImage	:	ITcVnImage;	(* Destination image *)
	END_VAR
	VAR_IN_OUT
		aColor	:	TcVnVector4_LREAL;	(* Color *)
	END_VAR
	VAR_INPUT
		nThickness	:	DINT;	(* Line thickness (if negative, the shape is filled) *)
		bIsClosed	:	BOOL;	(* If it is true, the function draws a line from the last point to the first point to close the polygon. *)
		eLineType	:	ETcVnLineType;	(* Line type *)
		nShift	:	UDINT;	(* Fractional bits of the coordinates (bit shift) *)
		hrPrev	:	HRESULT;	(* HRESULT indicating the result of previous operations (If SUCCEEDED(hrPrev) equals false, no operation is executed.) *)
	END_VAR

END_FUNCTION

// Functions/Drawing/F_VN_DrawRectangle

	{attribute 'TcIecLibraryType'}
	{attribute 'external_name' := 'F_VN_DrawRectangle_GUID_559B3717_92FE_4DE6_F2DA_D23616D7B583'}
	(* Draw a rectangle. *)
	FUNCTION F_VN_DrawRectangle : HRESULT
	VAR_INPUT
		nTopLeftX	:	UDINT;	(* x coordinate of the top left corner *)
		nTopLeftY	:	UDINT;	(* y coordinate of the top left corner *)
		nBottomRightX	:	UDINT;	(* x coordinate of the bottom right corner *)
		nBottomRightY	:	UDINT;	(* y coordinate of the bottom right corner *)
		ipDestImage	:	ITcVnImage;	(* Destination image *)
	END_VAR
	VAR_IN_OUT
		aColor	:	TcVnVector4_LREAL;	(* Color *)
	END_VAR
	VAR_INPUT
		nThickness	:	DINT;	(* Line thickness (if negative, the rectangle is filled) *)
		hrPrev	:	HRESULT;	(* HRESULT indicating the result of previous operations (If SUCCEEDED(hrPrev) equals false, no operation is executed.) *)
	END_VAR

END_FUNCTION

// Functions/Drawing/F_VN_DrawRectangle_TcVnRectangle_DINT

	{attribute 'TcIecLibraryType'}
	{attribute 'external_name' := 'F_VN_DrawRectangle_TcVnRectangle_DINT_GUID_AA7817DD_7AF7_4DF4_C83C_D3B85C72B15A'}
	(* Draw a rectangle. *)
	FUNCTION F_VN_DrawRectangle_TcVnRectangle_DINT : HRESULT
	VAR_IN_OUT
		stRectangle	:	TcVnRectangle_DINT;	(* Rectangle to be drawn *)
	END_VAR
	VAR_INPUT
		ipDestImage	:	ITcVnImage;	(* Destination image *)
	END_VAR
	VAR_IN_OUT
		aColor	:	TcVnVector4_LREAL;	(* Color *)
	END_VAR
	VAR_INPUT
		nThickness	:	DINT;	(* Line thickness (if negative, the rectangle is filled) *)
		hrPrev	:	HRESULT;	(* HRESULT indicating the result of previous operations (If SUCCEEDED(hrPrev) equals false, no operation is executed.) *)
	END_VAR

END_FUNCTION

// Functions/Drawing/F_VN_DrawRectangle_TcVnRectangle_UDINT

	{attribute 'TcIecLibraryType'}
	{attribute 'external_name' := 'F_VN_DrawRectangle_TcVnRectangle_UDINT_GUID_D49F1222_E68E_4F54_CC15_387AF19110AF'}
	(* Draw a rectangle. *)
	FUNCTION F_VN_DrawRectangle_TcVnRectangle_UDINT : HRESULT
	VAR_IN_OUT
		stRectangle	:	TcVnRectangle_UDINT;	(* Rectangle to be drawn *)
	END_VAR
	VAR_INPUT
		ipDestImage	:	ITcVnImage;	(* Destination image *)
	END_VAR
	VAR_IN_OUT
		aColor	:	TcVnVector4_LREAL;	(* Color *)
	END_VAR
	VAR_INPUT
		nThickness	:	DINT;	(* Line thickness (if negative, the rectangle is filled) *)
		hrPrev	:	HRESULT;	(* HRESULT indicating the result of previous operations (If SUCCEEDED(hrPrev) equals false, no operation is executed.) *)
	END_VAR

END_FUNCTION

// Functions/Drawing/F_VN_DrawRotatedRectangle

	{attribute 'TcIecLibraryType'}
	{attribute 'external_name' := 'F_VN_DrawRotatedRectangle_GUID_76F2F020_57B0_4942_FCCE_5DC3E4CE6220'}
	(* Draw a rectangle. *)
	FUNCTION F_VN_DrawRotatedRectangle : HRESULT
	VAR_IN_OUT
		stRectangle	:	TcVnRotatedRectangle;	(* Rectangle to be drawn (rotation angle in degrees) *)
	END_VAR
	VAR_INPUT
		ipDestImage	:	ITcVnImage;	(* Destination image *)
	END_VAR
	VAR_IN_OUT
		aColor	:	TcVnVector4_LREAL;	(* Color *)
	END_VAR
	VAR_INPUT
		nThickness	:	DINT;	(* Line thickness (if negative, the rectangle is filled) *)
		hrPrev	:	HRESULT;	(* HRESULT indicating the result of previous operations (If SUCCEEDED(hrPrev) equals false, no operation is executed.) *)
	END_VAR

END_FUNCTION

// Functions/Drawing/F_VN_DrawRotatedRectangleExp

	{attribute 'TcIecLibraryType'}
	{attribute 'external_name' := 'F_VN_DrawRotatedRectangleExp_GUID_61EBDDA5_AFA1_44BF_F771_7E4A9C1D02F4'}
	(* Draw a rectangle. (expert function) *)
	FUNCTION F_VN_DrawRotatedRectangleExp : HRESULT
	VAR_IN_OUT
		stRectangle	:	TcVnRotatedRectangle;	(* Rectangle to be drawn (rotation angle in degrees) *)
	END_VAR
	VAR_INPUT
		ipDestImage	:	ITcVnImage;	(* Destination image *)
	END_VAR
	VAR_IN_OUT
		aColor	:	TcVnVector4_LREAL;	(* Color *)
	END_VAR
	VAR_INPUT
		nThickness	:	DINT;	(* Line thickness (if negative, the rectangle is filled) *)
		eLineType	:	ETcVnLineType;	(* Line type *)
		hrPrev	:	HRESULT;	(* HRESULT indicating the result of previous operations (If SUCCEEDED(hrPrev) equals false, no operation is executed.) *)
	END_VAR

END_FUNCTION

// Functions/Drawing/F_VN_FillCircle

	{attribute 'TcIecLibraryType'}
	{attribute 'external_name' := 'F_VN_FillCircle_GUID_C81A317B_D294_4DD2_CFB7_83B48C61A946'}
	(* Paint a filled circle. *)
	FUNCTION F_VN_FillCircle : HRESULT
	VAR_INPUT
		nCenterX	:	UDINT;	(* x coordinate of the center *)
		nCenterY	:	UDINT;	(* y coordinate of the center *)
		nRadius	:	UDINT;	(* Radius *)
		ipDestImage	:	ITcVnImage;	(* Destination image *)
	END_VAR
	VAR_IN_OUT
		aColor	:	TcVnVector4_LREAL;	(* Color *)
	END_VAR
	VAR_INPUT
		hrPrev	:	HRESULT;	(* HRESULT indicating the result of previous operations (If SUCCEEDED(hrPrev) equals false, no operation is executed.) *)
	END_VAR

END_FUNCTION

// Functions/Drawing/F_VN_FillContours

	{attribute 'TcIecLibraryType'}
	{attribute 'external_name' := 'F_VN_FillContours_GUID_05FAC253_30FD_43F7_FD61_28FC729DA275'}
	(* Paint a single point set or multiple point sets that are interpreted as contours. *)
	FUNCTION F_VN_FillContours : HRESULT
	VAR_INPUT
		ipContours	:	ITcVnContainer;	(* Single contour (ContainerType_Vector_TcVnPoint2_DINT) or multiple contours (ContainerType_Vector_Vector_TcVnPoint2_DINT) *)
		nContourIndex	:	DINT;	(* Index of a specific contour to be drawn (if negative, all contours within the container are drawn) *)
		ipDestImage	:	ITcVnImage;	(* Destination image *)
	END_VAR
	VAR_IN_OUT
		aColor	:	TcVnVector4_LREAL;	(* Color *)
	END_VAR
	VAR_INPUT
		hrPrev	:	HRESULT;	(* HRESULT indicating the result of previous operations (If SUCCEEDED(hrPrev) equals false, no operation is executed.) *)
	END_VAR

END_FUNCTION

// Functions/Drawing/F_VN_FillEllipse

	{attribute 'TcIecLibraryType'}
	{attribute 'external_name' := 'F_VN_FillEllipse_GUID_C3348A8F_BDEF_485D_F618_232D2B13F77F'}
	(* Paint a filled ellipse. *)
	FUNCTION F_VN_FillEllipse : HRESULT
	VAR_IN_OUT
		stEllipse	:	TcVnRotatedRectangle;	(* Ellipse to be painted (rotation angle in degrees) *)
	END_VAR
	VAR_INPUT
		ipDestImage	:	ITcVnImage;	(* Destination image *)
	END_VAR
	VAR_IN_OUT
		aColor	:	TcVnVector4_LREAL;	(* Color *)
	END_VAR
	VAR_INPUT
		hrPrev	:	HRESULT;	(* HRESULT indicating the result of previous operations (If SUCCEEDED(hrPrev) equals false, no operation is executed.) *)
	END_VAR

END_FUNCTION

// Functions/Drawing/F_VN_FillPolygon

	{attribute 'TcIecLibraryType'}
	{attribute 'external_name' := 'F_VN_FillPolygon_GUID_BA26F71C_3F54_48B7_ECED_BE84CA809F66'}
	(* Paint a filled pologon using a set of points. *)
	FUNCTION F_VN_FillPolygon : HRESULT
	VAR_INPUT
		ipPoints	:	ITcVnContainer;	(* Container with TcVnPoint2_DINT, TcVnPoint2_REAL, or TcVnPoint2_LREAL elements *)
		ipDestImage	:	ITcVnImage;	(* Destination image *)
	END_VAR
	VAR_IN_OUT
		aColor	:	TcVnVector4_LREAL;	(* Color *)
	END_VAR
	VAR_INPUT
		hrPrev	:	HRESULT;	(* HRESULT indicating the result of previous operations (If SUCCEEDED(hrPrev) equals false, no operation is executed.) *)
	END_VAR

END_FUNCTION

// Functions/Drawing/F_VN_FillRectangle

	{attribute 'TcIecLibraryType'}
	{attribute 'external_name' := 'F_VN_FillRectangle_GUID_291B56A1_6B53_4DB0_CAAB_308F3DF1CF46'}
	(* Paint a filled rectangle. *)
	FUNCTION F_VN_FillRectangle : HRESULT
	VAR_INPUT
		nTopLeftX	:	UDINT;	(* x coordinate of the top left corner *)
		nTopLeftY	:	UDINT;	(* y coordinate of the top left corner *)
		nBottomRightX	:	UDINT;	(* x coordinate of the bottom right corner *)
		nBottomRightY	:	UDINT;	(* y coordinate of the bottom right corner *)
		ipDestImage	:	ITcVnImage;	(* Destination image *)
	END_VAR
	VAR_IN_OUT
		aColor	:	TcVnVector4_LREAL;	(* Color *)
	END_VAR
	VAR_INPUT
		hrPrev	:	HRESULT;	(* HRESULT indicating the result of previous operations (If SUCCEEDED(hrPrev) equals false, no operation is executed.) *)
	END_VAR

END_FUNCTION

// Functions/Drawing/F_VN_FillRotatedRectangle

	{attribute 'TcIecLibraryType'}
	{attribute 'external_name' := 'F_VN_FillRotatedRectangle_GUID_9AF68941_631E_4F53_F698_97DD38905251'}
	(* Paint a filled rectangle. *)
	FUNCTION F_VN_FillRotatedRectangle : HRESULT
	VAR_IN_OUT
		stRectangle	:	TcVnRotatedRectangle;	(* Rectangle to be painted (rotation angle in degrees) *)
	END_VAR
	VAR_INPUT
		ipDestImage	:	ITcVnImage;	(* Destination image *)
	END_VAR
	VAR_IN_OUT
		aColor	:	TcVnVector4_LREAL;	(* Color *)
	END_VAR
	VAR_INPUT
		hrPrev	:	HRESULT;	(* HRESULT indicating the result of previous operations (If SUCCEEDED(hrPrev) equals false, no operation is executed.) *)
	END_VAR

END_FUNCTION

// Functions/Drawing/F_VN_PlotIntensityProfile

	{attribute 'TcIecLibraryType'}
	{attribute 'external_name' := 'F_VN_PlotIntensityProfile_GUID_2D4D5FEC_E5E8_4313_EEEB_73F8D24DEEEC'}
	(* Plots the pixel intensity profile along a line segment in an image. *)
	FUNCTION F_VN_PlotIntensityProfile : HRESULT
	VAR_INPUT
		ipSrcImage	:	ITcVnImage;	(* Source image (USINT, 1 channel) *)
		ipDestImage	:	REFERENCE TO ITcVnImage;	(* Destination image (USINT, 1 channel. x: position, y: intensity, origin: bottom left. An appropriate destination image will be created if required.) *)
	END_VAR
	VAR_IN_OUT
		aStartPoint	:	TcVnPoint2_REAL;	(* Start point of the line segment *)
		aEndPoint	:	TcVnPoint2_REAL;	(* End point of the line segment *)
	END_VAR
	VAR_INPUT
		hrPrev	:	HRESULT;	(* HRESULT indicating the result of previous operations (If SUCCEEDED(hrPrev) equals false, no operation is executed.) *)
	END_VAR

END_FUNCTION

// Functions/Drawing/F_VN_PlotIntensityProfileExp

	{attribute 'TcIecLibraryType'}
	{attribute 'external_name' := 'F_VN_PlotIntensityProfileExp_GUID_873131B5_9D66_44BF_FD69_BD7E01FF51FE'}
	(* Plots the pixel intensity profile along a line segment in an image. (expert function) *)
	FUNCTION F_VN_PlotIntensityProfileExp : HRESULT
	VAR_INPUT
		ipSrcImage	:	ITcVnImage;	(* Source image (USINT, 1 channel) *)
		ipDestImage	:	REFERENCE TO ITcVnImage;	(* Destination image (USINT, 1 channel. x: position, y: intensity, origin: bottom left. An appropriate destination image will be created if required.) *)
	END_VAR
	VAR_IN_OUT
		aStartPoint	:	TcVnPoint2_REAL;	(* Start point of the line segment *)
		aEndPoint	:	TcVnPoint2_REAL;	(* End point of the line segment *)
		aBackgroundColor	:	TcVnVector4_LREAL;	(* Background color *)
		aLineColor	:	TcVnVector4_LREAL;	(* Line color *)
		aGridColor	:	TcVnVector4_LREAL;	(* Grid color *)
	END_VAR
	VAR_INPUT
		nScaleX	:	DINT;	(* Scale in x direction (ipDestImage will have a width of nScaleX * (ipSrcImage width - 1) + 1) *)
		nScaleY	:	DINT;	(* Scale in y direction (ipDestImage will have a height of nScaleY * 255 + 1) *)
		nThickness	:	DINT;	(* Line thickness *)
		nDestChannels	:	DINT;	(* ipDestImage channels (1 or 3) *)
		hrPrev	:	HRESULT;	(* HRESULT indicating the result of previous operations (If SUCCEEDED(hrPrev) equals false, no operation is executed.) *)
	END_VAR

END_FUNCTION

// Functions/Drawing/F_VN_PutLabel

	{attribute 'TcIecLibraryType'}
	{attribute 'external_name' := 'F_VN_PutLabel_GUID_33CC27F0_6B91_4CB7_F3EB_58ABDB7F3353'}
	(* Write a label (black text on white background) into an image. *)
	FUNCTION F_VN_PutLabel : HRESULT
	VAR_IN_OUT CONSTANT
		sText	:	STRING;	(* Text *)
	END_VAR
	VAR_INPUT
		ipDestImage	:	ITcVnImage;	(* Destination image *)
		nX	:	UDINT;	(* x coordinate (bottom left) *)
		nY	:	UDINT;	(* y coordinate (bottom left) *)
		fFontScale	:	LREAL;	(* Scaling factor *)
		hrPrev	:	HRESULT;	(* HRESULT indicating the result of previous operations (If SUCCEEDED(hrPrev) equals false, no operation is executed.) *)
	END_VAR

END_FUNCTION

// Functions/Drawing/F_VN_PutLabelExp

	{attribute 'TcIecLibraryType'}
	{attribute 'external_name' := 'F_VN_PutLabelExp_GUID_BD384753_AD6A_4D37_D566_0DDC7E7B3510'}
	(* Write a label (text on unified background) into an image. (expert function) *)
	FUNCTION F_VN_PutLabelExp : HRESULT
	VAR_IN_OUT CONSTANT
		sText	:	STRING;	(* Text *)
	END_VAR
	VAR_INPUT
		ipDestImage	:	ITcVnImage;	(* Destination image *)
		nX	:	UDINT;	(* x coordinate (bottom left) *)
		nY	:	UDINT;	(* y coordinate (bottom left) *)
		fFontScale	:	LREAL;	(* Scaling factor *)
		nThickness	:	UDINT;	(* Line thickness *)
		eFontType	:	ETcVnFontType;	(* Font type *)
	END_VAR
	VAR_IN_OUT
		aFontColor	:	TcVnVector4_LREAL;	(* Font color *)
		aBackgroundColor	:	TcVnVector4_LREAL;	(* Background color *)
	END_VAR
	VAR_INPUT
		eLineType	:	ETcVnLineType;	(* Line type *)
		hrPrev	:	HRESULT;	(* HRESULT indicating the result of previous operations (If SUCCEEDED(hrPrev) equals false, no operation is executed.) *)
	END_VAR

END_FUNCTION

// Functions/Drawing/F_VN_PutText

	{attribute 'TcIecLibraryType'}
	{attribute 'external_name' := 'F_VN_PutText_GUID_15696C1A_A437_43E9_F235_B76EB3182853'}
	(* Write text into an image. *)
	FUNCTION F_VN_PutText : HRESULT
	VAR_IN_OUT CONSTANT
		sText	:	STRING;	(* Text *)
	END_VAR
	VAR_INPUT
		ipDestImage	:	ITcVnImage;	(* Destination image *)
		nX	:	UDINT;	(* x coordinate (bottom left) *)
		nY	:	UDINT;	(* y coordinate (bottom left) *)
		eFontType	:	ETcVnFontType;	(* Font type *)
		fFontScale	:	LREAL;	(* Scaling factor *)
	END_VAR
	VAR_IN_OUT
		aColor	:	TcVnVector4_LREAL;	(* Text color *)
	END_VAR
	VAR_INPUT
		hrPrev	:	HRESULT;	(* HRESULT indicating the result of previous operations (If SUCCEEDED(hrPrev) equals false, no operation is executed.) *)
	END_VAR

END_FUNCTION

// Functions/Drawing/F_VN_PutTextExp

	{attribute 'TcIecLibraryType'}
	{attribute 'external_name' := 'F_VN_PutTextExp_GUID_4760069D_C695_4D3E_CE5F_BBBE94358E79'}
	(* Write text into an image. (expert function) *)
	FUNCTION F_VN_PutTextExp : HRESULT
	VAR_IN_OUT CONSTANT
		sText	:	STRING;	(* Text *)
	END_VAR
	VAR_INPUT
		ipDestImage	:	ITcVnImage;	(* Destination image *)
		nX	:	UDINT;	(* x coordinate (bottom left) *)
		nY	:	UDINT;	(* y coordinate (bottom left) *)
		eFontType	:	ETcVnFontType;	(* Font type *)
		fFontScale	:	LREAL;	(* Scaling factor *)
	END_VAR
	VAR_IN_OUT
		aColor	:	TcVnVector4_LREAL;	(* Text color *)
	END_VAR
	VAR_INPUT
		nThickness	:	DINT;	(* Line thickness *)
		eLineType	:	ETcVnLineType;	(* Line type *)
		bBottomLeftOrigin	:	BOOL;	(* Sets the image origin to the bottom left corner, if true *)
		hrPrev	:	HRESULT;	(* HRESULT indicating the result of previous operations (If SUCCEEDED(hrPrev) equals false, no operation is executed.) *)
	END_VAR

END_FUNCTION

// Functions/Keypoint Features/F_VN_FilterGoodMatches

	{attribute 'TcIecLibraryType'}
	{attribute 'external_name' := 'F_VN_FilterGoodMatches_GUID_804D23F3_118F_48F1_DD74_E35BD5CE1E7B'}
	(* Filter the descriptor matches and return only good ones. *)
	FUNCTION F_VN_FilterGoodMatches : HRESULT
	VAR_INPUT
		ipMatches	:	ITcVnContainer;	(* Container with descriptor matches (ContainerType_Vector_TcVnDMatch or ContainerType_Vector_Vector_TcVnDMatch) *)
		ipGoodMatches	:	REFERENCE TO ITcVnContainer;	(* Returns a container with good matches (ContainerType_Vector_TcVnDMatch) *)
		fMaxDist	:	REAL;	(* Maximum allowed descriptor distance (-1 disables this filter criterion) *)
		fMaxKnnRatio	:	REAL;	(* Maximum allowed distance ratio between first and second best match ([0..1], used for knn match results only, -1 disables this filter criterion) *)
		hrPrev	:	HRESULT;	(* HRESULT indicating the result of previous operations (If SUCCEEDED(hrPrev) equals false, no operation is executed.) *)
	END_VAR

END_FUNCTION

// Functions/Keypoint Features/F_VN_FindReferenceKeyPointsInImage

	{attribute 'TcIecLibraryType'}
	{attribute 'external_name' := 'F_VN_FindReferenceKeyPointsInImage_GUID_8114A7BB_3A23_4E9E_C4EA_31E98D46FE55'}
	(* Searches a reference image, represented by its keypoints and corresponding descriptors, in a given source image. *)
	FUNCTION F_VN_FindReferenceKeyPointsInImage : HRESULT
	VAR_INPUT
		ipSrcKeyPoints	:	ITcVnContainer;	(* KeyPoints of the source image, e.g. (ContainerType_Vector_TcVnKeyPoint) *)
		ipSrcDescriptors	:	ITcVnImage;	(* Descriptors of the source image KeyPoints *)
		ipRefKeyPoints	:	ITcVnContainer;	(* KeyPoints of the reference image, e.g. (ContainerType_Vector_TcVnKeyPoint) *)
		ipRefDescriptors	:	ITcVnImage;	(* Descriptors of the reference image KeyPoints *)
		nRefImageWidth	:	UDINT;	(* Width of the reference image in pixels *)
		nRefImageHeight	:	UDINT;	(* Height of the reference image in pixels *)
		ipEdgePoints	:	REFERENCE TO ITcVnContainer;	(* Returns a container with the 4 edge points of the reference image transformed into the coordinates of the source image (ContainerType_Vector_TcVnPoint2_REAL) *)
		fMaxDist	:	REAL;	(* Maximum allowed descriptor distance (-1 disables this filter criterion) *)
		fMaxKnnRatio	:	REAL;	(* Maximum allowed distance ratio between first and second best match ([0..1], -1 disables this filter criterion) *)
		eNormType	:	ETcVnNormalizationType;	(* Normalization type used for descriptor matching (HAMMING recommended for AKAZE, ORB, and BRISK. HAMMING2 is recommended for ORB if the ORB nBriefPoints parameter is 3 or 4. ) *)
		hrPrev	:	HRESULT;	(* HRESULT indicating the result of previous operations (If SUCCEEDED(hrPrev) equals false, no operation is executed.) *)
	END_VAR
	VAR_OUTPUT
		aPerspectiveTransform	:	TcVnMatrix3x3_LREAL;	(* Returns the perspective transformation matrix, which transforms the reference points to the source points *)
		nNumberOfGoodMatches	:	UDINT;	(* Return the number of good matches *)
		nNumberOfInliers	:	UDINT;	(* Return the number of inlier matches *)
	END_VAR

END_FUNCTION

// Functions/Keypoint Features/F_VN_FindReferenceKeyPointsInImageExp

	{attribute 'TcIecLibraryType'}
	{attribute 'external_name' := 'F_VN_FindReferenceKeyPointsInImageExp_GUID_C5775864_10D6_4E5A_F87E_703B262F2647'}
	(* Searches a reference image, represented by its keypoints and corresponding descriptors, in a given source image. (expert function) *)
	FUNCTION F_VN_FindReferenceKeyPointsInImageExp : HRESULT
	VAR_INPUT
		ipSrcKeyPoints	:	ITcVnContainer;	(* KeyPoints of the source image, e.g. (ContainerType_Vector_TcVnKeyPoint) *)
		ipSrcDescriptors	:	ITcVnImage;	(* Descriptors of the source image KeyPoints *)
		ipRefKeyPoints	:	ITcVnContainer;	(* KeyPoints of the reference image (ContainerType_Vector_TcVnKeyPoint) *)
		ipRefDescriptors	:	ITcVnImage;	(* Descriptors of the reference image KeyPoints *)
		nRefImageWidth	:	UDINT;	(* Width of the reference image in pixels *)
		nRefImageHeight	:	UDINT;	(* Height of the reference image in pixels *)
		ipEdgePoints	:	REFERENCE TO ITcVnContainer;	(* Returns a container with the 4 edge points of the reference image transformed into the coordinates of the source image (ContainerType_Vector_TcVnPoint2_REAL) *)
		fMaxDist	:	REAL;	(* Maximum allowed descriptor distance (-1 disables this filter criterion) *)
		fMaxKnnRatio	:	REAL;	(* Maximum allowed distance ratio between first and second best match ([0..1], -1 disables this filter criterion) *)
		eNormType	:	ETcVnNormalizationType;	(* Normalization type used for descriptor matching (HAMMING recommended for AKAZE, ORB, and BRISK. HAMMING2 is recommended for ORB if the ORB nBriefPoints parameter is 3 or 4. ) *)
		eAlgorithm	:	ETcVnEstimationAlgorithm;	(* Estimation algorithm used for computing the perspective transformation between the two point sets *)
		fReprojThreshold	:	LREAL;	(* Maximum allowed reprojection error to treat a point pair as an inlier (only used if eAlgorithm is RANSAC, RHO) *)
		nMaxIterations	:	UDINT;	(* Maximum number of RANSAC iterations *)
		fConfidence	:	LREAL;	(* Confidence (0..1) *)
		ipGoodMatches	:	REFERENCE TO ITcVnContainer;	(* Returns a container with good matches (optional, set to 0 if not required; ContainerType_Vector_TcVnDMatch) *)
		ipInlierMask	:	REFERENCE TO ITcVnContainer;	(* Returns a mask marking the inliers (optional, set to 0 if not required; ContainerType_Vector_SINT; only for RANSAC, LMEDS) *)
		hrPrev	:	HRESULT;	(* HRESULT indicating the result of previous operations (If SUCCEEDED(hrPrev) equals false, no operation is executed.) *)
	END_VAR
	VAR_OUTPUT
		aPerspectiveTransform	:	TcVnMatrix3x3_LREAL;	(* Returns the perspective transformation matrix, which transforms the reference points to the source points  *)
		nNumberOfGoodMatches	:	UDINT;	(* Return the number of good matches *)
		nNumberOfInliers	:	UDINT;	(* Return the number of inlier matches *)
	END_VAR

END_FUNCTION

